    // Event "A_zdown_c_on".
    IF NOT progress THEN
        b1 := (state0.dvar_M_sup_A_zdown) = (elit_Off);
        b1 := b1 AND ((state0.dvar_M_sup_sup) = (elit_X));
        IF b1 THEN
            b3 := (state0.dvar_M_sup_A_x2distributing) = (elit_On);
            b3 := b3 AND ((state0.dvar_M_sup_A_x2testing) = (elit_On));
            b3 := b3 AND ((state0.dvar_M_sup_S_Hinitialized) = (elit_On));
            b3 := b3 AND ((state0.dvar_M_sup_S_product4) = (elit_On));
            b3 := b3 AND ((state0.dvar_M_sup_S_product1) = (elit_On));
            b3 := b3 AND ((state0.dvar_M_sup_S_product2) = (elit_On));
            b3 := b3 AND ((state0.dvar_M_sup_S_product3) = (elit_On));
            b3 := b3 AND ((state0.dvar_M_sup_S_gripper) = (elit_Off));
            b3 := b3 AND ((state0.dvar_M_sup_S_xpos_at3) = (elit_On));
            b3 := b3 AND ((state0.dvar_M_sup_S_zpos_atup) = (elit_On));
            b2 := b3;
            IF NOT(b2) THEN
                b3 := (state0.dvar_M_sup_A_x2distributing) = (elit_On);
                b3 := b3 AND ((state0.dvar_M_sup_A_x2testing) = (elit_On));
                b3 := b3 AND ((state0.dvar_M_sup_S_Hinitialized) = (elit_On));
                b3 := b3 AND ((state0.dvar_M_sup_S_product4) = (elit_On));
                b3 := b3 AND ((state0.dvar_M_sup_S_product1) = (elit_On));
                b3 := b3 AND ((state0.dvar_M_sup_S_product2) = (elit_On));
                b3 := b3 AND ((state0.dvar_M_sup_S_product3) = (elit_On));
                b3 := b3 AND ((state0.dvar_M_sup_S_gripper) = (elit_Off));
                b3 := b3 AND ((state0.dvar_M_sup_S_xpos_at3) = (elit_Off));
                b3 := b3 AND ((state0.dvar_M_sup_S_xpos_at2) = (elit_On));
                b3 := b3 AND ((state0.dvar_M_sup_S_zpos_atup) = (elit_On));
                b2 := b2 OR (b3);
            END_IF;
            IF NOT(b2) THEN
                b3 := (state0.dvar_M_sup_A_x2distributing) = (elit_On);
                b3 := b3 AND ((state0.dvar_M_sup_A_x2testing) = (elit_On));
                b3 := b3 AND ((state0.dvar_M_sup_S_Hinitialized) = (elit_On));
                b3 := b3 AND ((state0.dvar_M_sup_S_product4) = (elit_On));
                b3 := b3 AND ((state0.dvar_M_sup_S_product1) = (elit_On));
                b3 := b3 AND ((state0.dvar_M_sup_S_product2) = (elit_On));
                b3 := b3 AND ((state0.dvar_M_sup_S_product3) = (elit_On));
                b3 := b3 AND ((state0.dvar_M_sup_S_gripper) = (elit_Off));
                b3 := b3 AND ((state0.dvar_M_sup_S_xpos_at3) = (elit_Off));
                b3 := b3 AND ((state0.dvar_M_sup_S_xpos_at2) = (elit_Off));
                b3 := b3 AND ((state0.dvar_M_sup_S_xpos_at1) = (elit_On));
                b3 := b3 AND ((state0.dvar_M_sup_S_zpos_atup) = (elit_On));
                b2 := b2 OR (b3);
            END_IF;
            IF NOT(b2) THEN
                b3 := (state0.dvar_M_sup_A_x2distributing) = (elit_On);
                b3 := b3 AND ((state0.dvar_M_sup_A_x2testing) = (elit_On));
                b3 := b3 AND ((state0.dvar_M_sup_S_Hinitialized) = (elit_On));
                b3 := b3 AND ((state0.dvar_M_sup_S_product4) = (elit_On));
                b3 := b3 AND ((state0.dvar_M_sup_S_product1) = (elit_On));
                b3 := b3 AND ((state0.dvar_M_sup_S_product2) = (elit_On));
                b3 := b3 AND ((state0.dvar_M_sup_S_product3) = (elit_Off));
                b3 := b3 AND ((state0.dvar_M_sup_S_gripper) = (elit_Off));
                b3 := b3 AND ((state0.dvar_M_sup_S_xpos_at2) = (elit_On));
                b3 := b3 AND ((state0.dvar_M_sup_S_zpos_atup) = (elit_On));
                b2 := b2 OR (b3);
            END_IF;
            IF NOT(b2) THEN
                b3 := (state0.dvar_M_sup_A_x2distributing) = (elit_On);
                b3 := b3 AND ((state0.dvar_M_sup_A_x2testing) = (elit_On));
                b3 := b3 AND ((state0.dvar_M_sup_S_Hinitialized) = (elit_On));
                b3 := b3 AND ((state0.dvar_M_sup_S_product4) = (elit_On));
                b3 := b3 AND ((state0.dvar_M_sup_S_product1) = (elit_On));
                b3 := b3 AND ((state0.dvar_M_sup_S_product2) = (elit_On));
                b3 := b3 AND ((state0.dvar_M_sup_S_product3) = (elit_Off));
                b3 := b3 AND ((state0.dvar_M_sup_S_gripper) = (elit_Off));
                b3 := b3 AND ((state0.dvar_M_sup_S_xpos_at2) = (elit_Off));
                b3 := b3 AND ((state0.dvar_M_sup_S_xpos_at1) = (elit_On));
                b3 := b3 AND ((state0.dvar_M_sup_S_zpos_atup) = (elit_On));
                b2 := b2 OR (b3);
            END_IF;
            IF NOT(b2) THEN
                b3 := (state0.dvar_M_sup_A_x2distributing) = (elit_On);
                b3 := b3 AND ((state0.dvar_M_sup_A_x2testing) = (elit_On));
                b3 := b3 AND ((state0.dvar_M_sup_S_Hinitialized) = (elit_On));
                b3 := b3 AND ((state0.dvar_M_sup_S_product4) = (elit_On));
                b3 := b3 AND ((state0.dvar_M_sup_S_product1) = (elit_On));
                b3 := b3 AND ((state0.dvar_M_sup_S_product2) = (elit_Off));
                b3 := b3 AND ((state0.dvar_M_sup_S_product3) = (elit_On));
                b3 := b3 AND ((state0.dvar_M_sup_S_gripper) = (elit_Off));
                b3 := b3 AND ((state0.dvar_M_sup_S_xpos_at3) = (elit_On));
                b3 := b3 AND ((state0.dvar_M_sup_S_zpos_atup) = (elit_On));
                b2 := b2 OR (b3);
            END_IF;
            IF NOT(b2) THEN
                b3 := (state0.dvar_M_sup_A_x2distributing) = (elit_On);
                b3 := b3 AND ((state0.dvar_M_sup_A_x2testing) = (elit_On));
                b3 := b3 AND ((state0.dvar_M_sup_S_Hinitialized) = (elit_On));
                b3 := b3 AND ((state0.dvar_M_sup_S_product4) = (elit_On));
                b3 := b3 AND ((state0.dvar_M_sup_S_product1) = (elit_On));
                b3 := b3 AND ((state0.dvar_M_sup_S_product2) = (elit_Off));
                b3 := b3 AND ((state0.dvar_M_sup_S_product3) = (elit_On));
                b3 := b3 AND ((state0.dvar_M_sup_S_gripper) = (elit_Off));
                b3 := b3 AND ((state0.dvar_M_sup_S_xpos_at3) = (elit_Off));
                b3 := b3 AND ((state0.dvar_M_sup_S_xpos_at1) = (elit_On));
                b3 := b3 AND ((state0.dvar_M_sup_S_zpos_atup) = (elit_On));
                b2 := b2 OR (b3);
            END_IF;
            IF NOT(b2) THEN
                b3 := (state0.dvar_M_sup_A_x2distributing) = (elit_On);
                b3 := b3 AND ((state0.dvar_M_sup_A_x2testing) = (elit_On));
                b3 := b3 AND ((state0.dvar_M_sup_S_Hinitialized) = (elit_On));
                b3 := b3 AND ((state0.dvar_M_sup_S_product4) = (elit_On));
                b3 := b3 AND ((state0.dvar_M_sup_S_product1) = (elit_On));
                b3 := b3 AND ((state0.dvar_M_sup_S_product2) = (elit_Off));
                b3 := b3 AND ((state0.dvar_M_sup_S_product3) = (elit_Off));
                b3 := b3 AND ((state0.dvar_M_sup_S_gripper) = (elit_Off));
                b3 := b3 AND ((state0.dvar_M_sup_S_xpos_at1) = (elit_On));
                b3 := b3 AND ((state0.dvar_M_sup_S_zpos_atup) = (elit_On));
                b2 := b2 OR (b3);
            END_IF;
            IF NOT(b2) THEN
                b3 := (state0.dvar_M_sup_A_x2distributing) = (elit_On);
                b3 := b3 AND ((state0.dvar_M_sup_A_x2testing) = (elit_On));
                b3 := b3 AND ((state0.dvar_M_sup_S_Hinitialized) = (elit_On));
                b3 := b3 AND ((state0.dvar_M_sup_S_product4) = (elit_On));
                b3 := b3 AND ((state0.dvar_M_sup_S_product1) = (elit_Off));
                b3 := b3 AND ((state0.dvar_M_sup_S_product2) = (elit_On));
                b3 := b3 AND ((state0.dvar_M_sup_S_product3) = (elit_On));
                b3 := b3 AND ((state0.dvar_M_sup_S_gripper) = (elit_Off));
                b3 := b3 AND ((state0.dvar_M_sup_S_xpos_at3) = (elit_On));
                b3 := b3 AND ((state0.dvar_M_sup_S_zpos_atup) = (elit_On));
                b2 := b2 OR (b3);
            END_IF;
            IF NOT(b2) THEN
                b3 := (state0.dvar_M_sup_A_x2distributing) = (elit_On);
                b3 := b3 AND ((state0.dvar_M_sup_A_x2testing) = (elit_On));
                b3 := b3 AND ((state0.dvar_M_sup_S_Hinitialized) = (elit_On));
                b3 := b3 AND ((state0.dvar_M_sup_S_product4) = (elit_On));
                b3 := b3 AND ((state0.dvar_M_sup_S_product1) = (elit_Off));
                b3 := b3 AND ((state0.dvar_M_sup_S_product2) = (elit_On));
                b3 := b3 AND ((state0.dvar_M_sup_S_product3) = (elit_On));
                b3 := b3 AND ((state0.dvar_M_sup_S_gripper) = (elit_Off));
                b3 := b3 AND ((state0.dvar_M_sup_S_xpos_at3) = (elit_Off));
                b3 := b3 AND ((state0.dvar_M_sup_S_xpos_at2) = (elit_On));
                b3 := b3 AND ((state0.dvar_M_sup_S_zpos_atup) = (elit_On));
                b2 := b2 OR (b3);
            END_IF;
            IF NOT(b2) THEN
                b3 := (state0.dvar_M_sup_A_x2distributing) = (elit_On);
                b3 := b3 AND ((state0.dvar_M_sup_A_x2testing) = (elit_On));
                b3 := b3 AND ((state0.dvar_M_sup_S_Hinitialized) = (elit_On));
                b3 := b3 AND ((state0.dvar_M_sup_S_product4) = (elit_On));
                b3 := b3 AND ((state0.dvar_M_sup_S_product1) = (elit_Off));
                b3 := b3 AND ((state0.dvar_M_sup_S_product2) = (elit_On));
                b3 := b3 AND ((state0.dvar_M_sup_S_product3) = (elit_Off));
                b3 := b3 AND ((state0.dvar_M_sup_S_gripper) = (elit_Off));
                b3 := b3 AND ((state0.dvar_M_sup_S_xpos_at2) = (elit_On));
                b3 := b3 AND ((state0.dvar_M_sup_S_zpos_atup) = (elit_On));
                b2 := b2 OR (b3);
            END_IF;
            IF NOT(b2) THEN
                b3 := (state0.dvar_M_sup_A_x2distributing) = (elit_On);
                b3 := b3 AND ((state0.dvar_M_sup_A_x2testing) = (elit_On));
                b3 := b3 AND ((state0.dvar_M_sup_S_Hinitialized) = (elit_On));
                b3 := b3 AND ((state0.dvar_M_sup_S_product4) = (elit_On));
                b3 := b3 AND ((state0.dvar_M_sup_S_product1) = (elit_Off));
                b3 := b3 AND ((state0.dvar_M_sup_S_product2) = (elit_Off));
                b3 := b3 AND ((state0.dvar_M_sup_S_product3) = (elit_On));
                b3 := b3 AND ((state0.dvar_M_sup_S_gripper) = (elit_Off));
                b3 := b3 AND ((state0.dvar_M_sup_S_xpos_at3) = (elit_On));
                b3 := b3 AND ((state0.dvar_M_sup_S_zpos_atup) = (elit_On));
                b2 := b2 OR (b3);
            END_IF;
            IF NOT(b2) THEN
                b3 := (state0.dvar_M_sup_A_x2distributing) = (elit_On);
                b3 := b3 AND ((state0.dvar_M_sup_A_x2testing) = (elit_On));
                b3 := b3 AND ((state0.dvar_M_sup_S_Hinitialized) = (elit_On));
                b3 := b3 AND ((state0.dvar_M_sup_S_product4) = (elit_Off));
                b3 := b3 AND ((state0.dvar_M_sup_S_product1) = (elit_On));
                b3 := b3 AND ((state0.dvar_M_sup_S_product2) = (elit_On));
                b3 := b3 AND ((state0.dvar_M_sup_S_product3) = (elit_On));
                b3 := b3 AND ((state0.dvar_M_sup_S_gripper) = (elit_On));
                b3 := b3 AND ((state0.dvar_M_sup_S_xpos_atdrop) = (elit_On));
                b3 := b3 AND ((state0.dvar_M_sup_S_zpos_atup) = (elit_On));
                b2 := b2 OR (b3);
            END_IF;
            IF NOT(b2) THEN
                b3 := (state0.dvar_M_sup_A_x2distributing) = (elit_On);
                b3 := b3 AND ((state0.dvar_M_sup_A_x2testing) = (elit_On));
                b3 := b3 AND ((state0.dvar_M_sup_S_Hinitialized) = (elit_On));
                b3 := b3 AND ((state0.dvar_M_sup_S_product4) = (elit_Off));
                b3 := b3 AND ((state0.dvar_M_sup_S_product1) = (elit_On));
                b3 := b3 AND ((state0.dvar_M_sup_S_product2) = (elit_On));
                b3 := b3 AND ((state0.dvar_M_sup_S_product3) = (elit_On));
                b3 := b3 AND ((state0.dvar_M_sup_S_gripper) = (elit_Off));
                b3 := b3 AND ((state0.dvar_M_sup_S_xpos_at3) = (elit_On));
                b3 := b3 AND ((state0.dvar_M_sup_S_zpos_atup) = (elit_On));
                b2 := b2 OR (b3);
            END_IF;
            IF NOT(b2) THEN
                b3 := (state0.dvar_M_sup_A_x2distributing) = (elit_On);
                b3 := b3 AND ((state0.dvar_M_sup_A_x2testing) = (elit_On));
                b3 := b3 AND ((state0.dvar_M_sup_S_Hinitialized) = (elit_On));
                b3 := b3 AND ((state0.dvar_M_sup_S_product4) = (elit_Off));
                b3 := b3 AND ((state0.dvar_M_sup_S_product1) = (elit_On));
                b3 := b3 AND ((state0.dvar_M_sup_S_product2) = (elit_On));
                b3 := b3 AND ((state0.dvar_M_sup_S_product3) = (elit_On));
                b3 := b3 AND ((state0.dvar_M_sup_S_gripper) = (elit_Off));
                b3 := b3 AND ((state0.dvar_M_sup_S_xpos_at3) = (elit_Off));
                b3 := b3 AND ((state0.dvar_M_sup_S_xpos_at2) = (elit_On));
                b3 := b3 AND ((state0.dvar_M_sup_S_zpos_atup) = (elit_On));
                b2 := b2 OR (b3);
            END_IF;
            IF NOT(b2) THEN
                b3 := (state0.dvar_M_sup_A_x2distributing) = (elit_On);
                b3 := b3 AND ((state0.dvar_M_sup_A_x2testing) = (elit_On));
                b3 := b3 AND ((state0.dvar_M_sup_S_Hinitialized) = (elit_On));
                b3 := b3 AND ((state0.dvar_M_sup_S_product4) = (elit_Off));
                b3 := b3 AND ((state0.dvar_M_sup_S_product1) = (elit_On));
                b3 := b3 AND ((state0.dvar_M_sup_S_product2) = (elit_On));
                b3 := b3 AND ((state0.dvar_M_sup_S_product3) = (elit_On));
                b3 := b3 AND ((state0.dvar_M_sup_S_gripper) = (elit_Off));
                b3 := b3 AND ((state0.dvar_M_sup_S_xpos_at3) = (elit_Off));
                b3 := b3 AND ((state0.dvar_M_sup_S_xpos_at2) = (elit_Off));
                b3 := b3 AND ((state0.dvar_M_sup_S_xpos_at1) = (elit_On));
                b3 := b3 AND ((state0.dvar_M_sup_S_zpos_atup) = (elit_On));
                b2 := b2 OR (b3);
            END_IF;
            IF NOT(b2) THEN
                b3 := (state0.dvar_M_sup_A_x2distributing) = (elit_On);
                b3 := b3 AND ((state0.dvar_M_sup_A_x2testing) = (elit_On));
                b3 := b3 AND ((state0.dvar_M_sup_S_Hinitialized) = (elit_On));
                b3 := b3 AND ((state0.dvar_M_sup_S_product4) = (elit_Off));
                b3 := b3 AND ((state0.dvar_M_sup_S_product1) = (elit_On));
                b3 := b3 AND ((state0.dvar_M_sup_S_product2) = (elit_On));
                b3 := b3 AND ((state0.dvar_M_sup_S_product3) = (elit_Off));
                b3 := b3 AND ((state0.dvar_M_sup_S_gripper) = (elit_On));
                b3 := b3 AND ((state0.dvar_M_sup_S_xpos_atdrop) = (elit_On));
                b3 := b3 AND ((state0.dvar_M_sup_S_zpos_atup) = (elit_On));
                b2 := b2 OR (b3);
            END_IF;
            IF NOT(b2) THEN
                b3 := (state0.dvar_M_sup_A_x2distributing) = (elit_On);
                b3 := b3 AND ((state0.dvar_M_sup_A_x2testing) = (elit_On));
                b3 := b3 AND ((state0.dvar_M_sup_S_Hinitialized) = (elit_On));
                b3 := b3 AND ((state0.dvar_M_sup_S_product4) = (elit_Off));
                b3 := b3 AND ((state0.dvar_M_sup_S_product1) = (elit_On));
                b3 := b3 AND ((state0.dvar_M_sup_S_product2) = (elit_On));
                b3 := b3 AND ((state0.dvar_M_sup_S_product3) = (elit_Off));
                b3 := b3 AND ((state0.dvar_M_sup_S_gripper) = (elit_Off));
                b3 := b3 AND ((state0.dvar_M_sup_S_xpos_at2) = (elit_On));
                b3 := b3 AND ((state0.dvar_M_sup_S_zpos_atup) = (elit_On));
                b2 := b2 OR (b3);
            END_IF;
            IF NOT(b2) THEN
                b3 := (state0.dvar_M_sup_A_x2distributing) = (elit_On);
                b3 := b3 AND ((state0.dvar_M_sup_A_x2testing) = (elit_On));
                b3 := b3 AND ((state0.dvar_M_sup_S_Hinitialized) = (elit_On));
                b3 := b3 AND ((state0.dvar_M_sup_S_product4) = (elit_Off));
                b3 := b3 AND ((state0.dvar_M_sup_S_product1) = (elit_On));
                b3 := b3 AND ((state0.dvar_M_sup_S_product2) = (elit_On));
                b3 := b3 AND ((state0.dvar_M_sup_S_product3) = (elit_Off));
                b3 := b3 AND ((state0.dvar_M_sup_S_gripper) = (elit_Off));
                b3 := b3 AND ((state0.dvar_M_sup_S_xpos_at2) = (elit_Off));
                b3 := b3 AND ((state0.dvar_M_sup_S_xpos_at1) = (elit_On));
                b3 := b3 AND ((state0.dvar_M_sup_S_zpos_atup) = (elit_On));
                b2 := b2 OR (b3);
            END_IF;
            IF NOT(b2) THEN
                b3 := (state0.dvar_M_sup_A_x2distributing) = (elit_On);
                b3 := b3 AND ((state0.dvar_M_sup_A_x2testing) = (elit_On));
                b3 := b3 AND ((state0.dvar_M_sup_S_Hinitialized) = (elit_On));
                b3 := b3 AND ((state0.dvar_M_sup_S_product4) = (elit_Off));
                b3 := b3 AND ((state0.dvar_M_sup_S_product1) = (elit_On));
                b3 := b3 AND ((state0.dvar_M_sup_S_product2) = (elit_Off));
                b3 := b3 AND ((state0.dvar_M_sup_S_product3) = (elit_On));
                b3 := b3 AND ((state0.dvar_M_sup_S_gripper) = (elit_On));
                b3 := b3 AND ((state0.dvar_M_sup_S_xpos_atdrop) = (elit_On));
                b3 := b3 AND ((state0.dvar_M_sup_S_zpos_atup) = (elit_On));
                b2 := b2 OR (b3);
            END_IF;
            IF NOT(b2) THEN
                b3 := (state0.dvar_M_sup_A_x2distributing) = (elit_On);
                b3 := b3 AND ((state0.dvar_M_sup_A_x2testing) = (elit_On));
                b3 := b3 AND ((state0.dvar_M_sup_S_Hinitialized) = (elit_On));
                b3 := b3 AND ((state0.dvar_M_sup_S_product4) = (elit_Off));
                b3 := b3 AND ((state0.dvar_M_sup_S_product1) = (elit_On));
                b3 := b3 AND ((state0.dvar_M_sup_S_product2) = (elit_Off));
                b3 := b3 AND ((state0.dvar_M_sup_S_product3) = (elit_On));
                b3 := b3 AND ((state0.dvar_M_sup_S_gripper) = (elit_Off));
                b3 := b3 AND ((state0.dvar_M_sup_S_xpos_at3) = (elit_On));
                b3 := b3 AND ((state0.dvar_M_sup_S_zpos_atup) = (elit_On));
                b2 := b2 OR (b3);
            END_IF;
            IF NOT(b2) THEN
                b3 := (state0.dvar_M_sup_A_x2distributing) = (elit_On);
                b3 := b3 AND ((state0.dvar_M_sup_A_x2testing) = (elit_On));
                b3 := b3 AND ((state0.dvar_M_sup_S_Hinitialized) = (elit_On));
                b3 := b3 AND ((state0.dvar_M_sup_S_product4) = (elit_Off));
                b3 := b3 AND ((state0.dvar_M_sup_S_product1) = (elit_On));
                b3 := b3 AND ((state0.dvar_M_sup_S_product2) = (elit_Off));
                b3 := b3 AND ((state0.dvar_M_sup_S_product3) = (elit_On));
                b3 := b3 AND ((state0.dvar_M_sup_S_gripper) = (elit_Off));
                b3 := b3 AND ((state0.dvar_M_sup_S_xpos_at3) = (elit_Off));
                b3 := b3 AND ((state0.dvar_M_sup_S_xpos_at1) = (elit_On));
                b3 := b3 AND ((state0.dvar_M_sup_S_zpos_atup) = (elit_On));
                b2 := b2 OR (b3);
            END_IF;
            IF NOT(b2) THEN
                b3 := (state0.dvar_M_sup_A_x2distributing) = (elit_On);
                b3 := b3 AND ((state0.dvar_M_sup_A_x2testing) = (elit_On));
                b3 := b3 AND ((state0.dvar_M_sup_S_Hinitialized) = (elit_On));
                b3 := b3 AND ((state0.dvar_M_sup_S_product4) = (elit_Off));
                b3 := b3 AND ((state0.dvar_M_sup_S_product1) = (elit_On));
                b3 := b3 AND ((state0.dvar_M_sup_S_product2) = (elit_Off));
                b3 := b3 AND ((state0.dvar_M_sup_S_product3) = (elit_Off));
                b3 := b3 AND ((state0.dvar_M_sup_S_gripper) = (elit_On));
                b3 := b3 AND ((state0.dvar_M_sup_S_xpos_atdrop) = (elit_On));
                b3 := b3 AND ((state0.dvar_M_sup_S_zpos_atup) = (elit_On));
                b2 := b2 OR (b3);
            END_IF;
            IF NOT(b2) THEN
                b3 := (state0.dvar_M_sup_A_x2distributing) = (elit_On);
                b3 := b3 AND ((state0.dvar_M_sup_A_x2testing) = (elit_On));
                b3 := b3 AND ((state0.dvar_M_sup_S_Hinitialized) = (elit_On));
                b3 := b3 AND ((state0.dvar_M_sup_S_product4) = (elit_Off));
                b3 := b3 AND ((state0.dvar_M_sup_S_product1) = (elit_On));
                b3 := b3 AND ((state0.dvar_M_sup_S_product2) = (elit_Off));
                b3 := b3 AND ((state0.dvar_M_sup_S_product3) = (elit_Off));
                b3 := b3 AND ((state0.dvar_M_sup_S_gripper) = (elit_Off));
                b3 := b3 AND ((state0.dvar_M_sup_S_xpos_at1) = (elit_On));
                b3 := b3 AND ((state0.dvar_M_sup_S_zpos_atup) = (elit_On));
                b2 := b2 OR (b3);
            END_IF;
            IF NOT(b2) THEN
                b3 := (state0.dvar_M_sup_A_x2distributing) = (elit_On);
                b3 := b3 AND ((state0.dvar_M_sup_A_x2testing) = (elit_On));
                b3 := b3 AND ((state0.dvar_M_sup_S_Hinitialized) = (elit_On));
                b3 := b3 AND ((state0.dvar_M_sup_S_product4) = (elit_Off));
                b3 := b3 AND ((state0.dvar_M_sup_S_product1) = (elit_Off));
                b3 := b3 AND ((state0.dvar_M_sup_S_product2) = (elit_On));
                b3 := b3 AND ((state0.dvar_M_sup_S_product3) = (elit_On));
                b3 := b3 AND ((state0.dvar_M_sup_S_gripper) = (elit_On));
                b3 := b3 AND ((state0.dvar_M_sup_S_xpos_atdrop) = (elit_On));
                b3 := b3 AND ((state0.dvar_M_sup_S_zpos_atup) = (elit_On));
                b2 := b2 OR (b3);
            END_IF;
            IF NOT(b2) THEN
                b3 := (state0.dvar_M_sup_A_x2distributing) = (elit_On);
                b3 := b3 AND ((state0.dvar_M_sup_A_x2testing) = (elit_On));
                b3 := b3 AND ((state0.dvar_M_sup_S_Hinitialized) = (elit_On));
                b3 := b3 AND ((state0.dvar_M_sup_S_product4) = (elit_Off));
                b3 := b3 AND ((state0.dvar_M_sup_S_product1) = (elit_Off));
                b3 := b3 AND ((state0.dvar_M_sup_S_product2) = (elit_On));
                b3 := b3 AND ((state0.dvar_M_sup_S_product3) = (elit_On));
                b3 := b3 AND ((state0.dvar_M_sup_S_gripper) = (elit_Off));
                b3 := b3 AND ((state0.dvar_M_sup_S_xpos_at3) = (elit_On));
                b3 := b3 AND ((state0.dvar_M_sup_S_zpos_atup) = (elit_On));
                b2 := b2 OR (b3);
            END_IF;
            IF NOT(b2) THEN
                b3 := (state0.dvar_M_sup_A_x2distributing) = (elit_On);
                b3 := b3 AND ((state0.dvar_M_sup_A_x2testing) = (elit_On));
                b3 := b3 AND ((state0.dvar_M_sup_S_Hinitialized) = (elit_On));
                b3 := b3 AND ((state0.dvar_M_sup_S_product4) = (elit_Off));
                b3 := b3 AND ((state0.dvar_M_sup_S_product1) = (elit_Off));
                b3 := b3 AND ((state0.dvar_M_sup_S_product2) = (elit_On));
                b3 := b3 AND ((state0.dvar_M_sup_S_product3) = (elit_On));
                b3 := b3 AND ((state0.dvar_M_sup_S_gripper) = (elit_Off));
                b3 := b3 AND ((state0.dvar_M_sup_S_xpos_at3) = (elit_Off));
                b3 := b3 AND ((state0.dvar_M_sup_S_xpos_at2) = (elit_On));
                b3 := b3 AND ((state0.dvar_M_sup_S_zpos_atup) = (elit_On));
                b2 := b2 OR (b3);
            END_IF;
            IF NOT(b2) THEN
                b3 := (state0.dvar_M_sup_A_x2distributing) = (elit_On);
                b3 := b3 AND ((state0.dvar_M_sup_A_x2testing) = (elit_On));
                b3 := b3 AND ((state0.dvar_M_sup_S_Hinitialized) = (elit_On));
                b3 := b3 AND ((state0.dvar_M_sup_S_product4) = (elit_Off));
                b3 := b3 AND ((state0.dvar_M_sup_S_product1) = (elit_Off));
                b3 := b3 AND ((state0.dvar_M_sup_S_product2) = (elit_On));
                b3 := b3 AND ((state0.dvar_M_sup_S_product3) = (elit_Off));
                b3 := b3 AND ((state0.dvar_M_sup_S_gripper) = (elit_On));
                b3 := b3 AND ((state0.dvar_M_sup_S_xpos_atdrop) = (elit_On));
                b3 := b3 AND ((state0.dvar_M_sup_S_zpos_atup) = (elit_On));
                b2 := b2 OR (b3);
            END_IF;
            IF NOT(b2) THEN
                b3 := (state0.dvar_M_sup_A_x2distributing) = (elit_On);
                b3 := b3 AND ((state0.dvar_M_sup_A_x2testing) = (elit_On));
                b3 := b3 AND ((state0.dvar_M_sup_S_Hinitialized) = (elit_On));
                b3 := b3 AND ((state0.dvar_M_sup_S_product4) = (elit_Off));
                b3 := b3 AND ((state0.dvar_M_sup_S_product1) = (elit_Off));
                b3 := b3 AND ((state0.dvar_M_sup_S_product2) = (elit_On));
                b3 := b3 AND ((state0.dvar_M_sup_S_product3) = (elit_Off));
                b3 := b3 AND ((state0.dvar_M_sup_S_gripper) = (elit_Off));
                b3 := b3 AND ((state0.dvar_M_sup_S_xpos_at2) = (elit_On));
                b3 := b3 AND ((state0.dvar_M_sup_S_zpos_atup) = (elit_On));
                b2 := b2 OR (b3);
            END_IF;
            IF NOT(b2) THEN
                b3 := (state0.dvar_M_sup_A_x2distributing) = (elit_On);
                b3 := b3 AND ((state0.dvar_M_sup_A_x2testing) = (elit_On));
                b3 := b3 AND ((state0.dvar_M_sup_S_Hinitialized) = (elit_On));
                b3 := b3 AND ((state0.dvar_M_sup_S_product4) = (elit_Off));
                b3 := b3 AND ((state0.dvar_M_sup_S_product1) = (elit_Off));
                b3 := b3 AND ((state0.dvar_M_sup_S_product2) = (elit_Off));
                b3 := b3 AND ((state0.dvar_M_sup_S_product3) = (elit_On));
                b3 := b3 AND ((state0.dvar_M_sup_S_gripper) = (elit_On));
                b3 := b3 AND ((state0.dvar_M_sup_S_xpos_atdrop) = (elit_On));
                b3 := b3 AND ((state0.dvar_M_sup_S_zpos_atup) = (elit_On));
                b2 := b2 OR (b3);
            END_IF;
            IF NOT(b2) THEN
                b3 := (state0.dvar_M_sup_A_x2distributing) = (elit_On);
                b3 := b3 AND ((state0.dvar_M_sup_A_x2testing) = (elit_On));
                b3 := b3 AND ((state0.dvar_M_sup_S_Hinitialized) = (elit_On));
                b3 := b3 AND ((state0.dvar_M_sup_S_product4) = (elit_Off));
                b3 := b3 AND ((state0.dvar_M_sup_S_product1) = (elit_Off));
                b3 := b3 AND ((state0.dvar_M_sup_S_product2) = (elit_Off));
                b3 := b3 AND ((state0.dvar_M_sup_S_product3) = (elit_On));
                b3 := b3 AND ((state0.dvar_M_sup_S_gripper) = (elit_Off));
                b3 := b3 AND ((state0.dvar_M_sup_S_xpos_at3) = (elit_On));
                b3 := b3 AND ((state0.dvar_M_sup_S_zpos_atup) = (elit_On));
                b2 := b2 OR (b3);
            END_IF;
            IF NOT(b2) THEN
                b3 := (state0.dvar_M_sup_A_x2distributing) = (elit_On);
                b3 := b3 AND ((state0.dvar_M_sup_A_x2testing) = (elit_On));
                b3 := b3 AND ((state0.dvar_M_sup_S_Hinitialized) = (elit_On));
                b3 := b3 AND ((state0.dvar_M_sup_S_product4) = (elit_Off));
                b3 := b3 AND ((state0.dvar_M_sup_S_product1) = (elit_Off));
                b3 := b3 AND ((state0.dvar_M_sup_S_product2) = (elit_Off));
                b3 := b3 AND ((state0.dvar_M_sup_S_product3) = (elit_Off));
                b3 := b3 AND ((state0.dvar_M_sup_S_gripper) = (elit_On));
                b3 := b3 AND ((state0.dvar_M_sup_S_xpos_atdrop) = (elit_On));
                b3 := b3 AND ((state0.dvar_M_sup_S_zpos_atup) = (elit_On));
                b2 := b2 OR (b3);
            END_IF;
            b1 := b1 AND (b2);
        END_IF;
        IF b1 THEN
            progress := TRUE;
            state1 := state0;

            state1.dvar_M_sup_A_zdown := elit_On;

            state0 := state1;
        END_IF;
    END_IF;

    // Event "BTimer_c_on".
    IF NOT progress THEN
        b1 := (state0.dvar_M_BTimer1) = (elit_Off);
        b1 := b1 AND ((state0.dvar_M_sup_BTimer) = (elit_Off));
        b1 := b1 AND ((state0.dvar_M_sup_sup) = (elit_X));
        b1 := b1 AND ((state0.dvar_M_sup_S_atend) = (elit_On));
        IF b1 THEN
            progress := TRUE;
            state1 := state0;

            state1.dvar_M_BTimer1 := elit_Running;
            state1.dvar_M_sup_BTimer := elit_Running;

            state0 := state1;
        END_IF;
    END_IF;

    // Event "BTimer_c_reset".
    IF NOT progress THEN
        b2 := (state0.dvar_M_BTimer1) = (elit_Running);
        b2 := b2 OR ((state0.dvar_M_BTimer1) = (elit_Timeout));
        b1 := b2;
        IF b1 THEN
            b2 := (state0.dvar_M_sup_BTimer) = (elit_Running);
            b2 := b2 OR ((state0.dvar_M_sup_BTimer) = (elit_Timeout));
            b1 := b1 AND (b2);
        END_IF;
        b1 := b1 AND ((state0.dvar_M_sup_sup) = (elit_X));
        IF b1 THEN
            b2 := (state0.dvar_M_sup_A_conveyerB) = (elit_Off);
            b2 := b2 OR ((state0.dvar_M_sup_S_atin) = (elit_On));
            b1 := b1 AND (b2);
        END_IF;
        IF b1 THEN
            progress := TRUE;
            state1 := state0;

            IF ((state0.dvar_M_BTimer1) = (elit_Running)) THEN
                state1.cvar_M_BTimer1_t := 0.0;
                state1.dvar_M_BTimer1 := elit_Off;
            ELSIF ((state0.dvar_M_BTimer1) = (elit_Timeout)) THEN
                state1.cvar_M_BTimer1_t := 0.0;
                state1.dvar_M_BTimer1 := elit_Off;
            END_IF;
            IF ((state0.dvar_M_sup_BTimer) = (elit_Running)) THEN
                state1.dvar_M_sup_BTimer := elit_Off;
            ELSIF ((state0.dvar_M_sup_BTimer) = (elit_Timeout)) THEN
                state1.dvar_M_sup_BTimer := elit_Off;
            END_IF;

            state0 := state1;
        END_IF;
    END_IF;

    // Event "BTimer_u_timeout".
    IF NOT progress THEN
        b1 := (state0.dvar_M_BTimer1) = (elit_Running);
        b1 := b1 AND ((state0.cvar_M_BTimer1_t) > (0.5));
        b1 := b1 AND ((state0.dvar_M_sup_BTimer) = (elit_Running));
        IF b1 THEN
            progress := TRUE;
            state1 := state0;

            state1.dvar_M_BTimer1 := elit_Timeout;
            state1.dvar_M_sup_BTimer := elit_Timeout;

            state0 := state1;
        END_IF;
    END_IF;

    // Event "S_atdrill_u_off".
    IF NOT progress THEN
        b1 := (state0.dvar_M_BoolToEventsP) = (elit_X);
        b1 := b1 AND (NOT(ivar_s_atdrill));
        b1 := b1 AND ((state0.dvar_M_sup_S_atdrill) = (elit_On));
        IF b1 THEN
            progress := TRUE;
            state1 := state0;

            state1.dvar_M_sup_S_atdrill := elit_Off;

            state0 := state1;
        END_IF;
    END_IF;

    // Event "S_atdrill_u_on".
    IF NOT progress THEN
        b1 := (state0.dvar_M_BoolToEventsP) = (elit_X);
        b1 := b1 AND (ivar_s_atdrill);
        b1 := b1 AND ((state0.dvar_M_sup_S_atdrill) = (elit_Off));
        IF b1 THEN
            progress := TRUE;
            state1 := state0;

            state1.dvar_M_sup_S_atdrill := elit_On;

            state0 := state1;
        END_IF;
    END_IF;

    // Event "S_atend_u_off".
    IF NOT progress THEN
        b1 := (state0.dvar_M_BoolToEventsTB) = (elit_X);
        b1 := b1 AND (NOT(ivar_s_atend));
        b1 := b1 AND ((state0.dvar_M_sup_S_atend) = (elit_On));
        IF b1 THEN
            progress := TRUE;
            state1 := state0;

            state1.dvar_M_sup_S_atend := elit_Off;

            state0 := state1;
        END_IF;
    END_IF;

    // Event "S_atend_u_on".
    IF NOT progress THEN
        b1 := (state0.dvar_M_BoolToEventsTB) = (elit_X);
        b1 := b1 AND (ivar_s_atend);
        b1 := b1 AND ((state0.dvar_M_sup_S_atend) = (elit_Off));
        IF b1 THEN
            progress := TRUE;
            state1 := state0;

            state1.dvar_M_sup_S_atend := elit_On;

            state0 := state1;
        END_IF;
    END_IF;

    // Event "S_atexit_u_off".
    IF NOT progress THEN
        b1 := (state0.dvar_M_BoolToEventsP) = (elit_X);
        b1 := b1 AND (NOT(ivar_s_atexit));
        b1 := b1 AND ((state0.dvar_M_sup_S_atexit) = (elit_On));
        IF b1 THEN
            progress := TRUE;
            state1 := state0;

            state1.dvar_M_sup_S_atexit := elit_Off;

            state0 := state1;
        END_IF;
    END_IF;

    // Event "S_atexit_u_on".
    IF NOT progress THEN
        b1 := (state0.dvar_M_BoolToEventsP) = (elit_X);
        b1 := b1 AND (ivar_s_atexit);
        b1 := b1 AND ((state0.dvar_M_sup_S_atexit) = (elit_Off));
        IF b1 THEN
            progress := TRUE;
            state1 := state0;

            state1.dvar_M_sup_S_atexit := elit_On;

            state0 := state1;
        END_IF;
    END_IF;

    // Event "S_atin_u_off".
    IF NOT progress THEN
        b1 := (state0.dvar_M_BoolToEventsTB) = (elit_X);
        b1 := b1 AND (NOT(ivar_s_atin));
        b1 := b1 AND ((state0.dvar_M_sup_S_atin) = (elit_On));
        IF b1 THEN
            progress := TRUE;
            state1 := state0;

            state1.dvar_M_sup_S_atin := elit_Off;

            state0 := state1;
        END_IF;
    END_IF;

    // Event "S_atin_u_on".
    IF NOT progress THEN
        b1 := (state0.dvar_M_BoolToEventsTB) = (elit_X);
        b1 := b1 AND (ivar_s_atin);
        b1 := b1 AND ((state0.dvar_M_sup_S_atin) = (elit_Off));
        IF b1 THEN
            progress := TRUE;
            state1 := state0;

            state1.dvar_M_sup_S_atin := elit_On;

            state0 := state1;
        END_IF;
    END_IF;

    // Event "S_atinput_u_off".
    IF NOT progress THEN
        b1 := (state0.dvar_M_BoolToEventsP) = (elit_X);
        b1 := b1 AND (NOT(ivar_s_atinput));
        b1 := b1 AND ((state0.dvar_M_sup_S_atinput) = (elit_On));
        IF b1 THEN
            progress := TRUE;
            state1 := state0;

            state1.dvar_M_sup_S_atinput := elit_Off;

            state0 := state1;
        END_IF;
    END_IF;

    // Event "S_atinput_u_on".
    IF NOT progress THEN
        b1 := (state0.dvar_M_BoolToEventsP) = (elit_X);
        b1 := b1 AND (ivar_s_atinput);
        b1 := b1 AND ((state0.dvar_M_sup_S_atinput) = (elit_Off));
        IF b1 THEN
            progress := TRUE;
            state1 := state0;

            state1.dvar_M_sup_S_atinput := elit_On;

            state0 := state1;
        END_IF;
    END_IF;

    // Event "S_atseparator_u_off".
    IF NOT progress THEN
        b1 := (state0.dvar_M_BoolToEventsTB) = (elit_X);
        b1 := b1 AND (NOT(ivar_s_atseparator));
        b1 := b1 AND ((state0.dvar_M_sup_S_atseparator) = (elit_On));
        IF b1 THEN
            progress := TRUE;
            state1 := state0;

            state1.dvar_M_sup_S_atseparator := elit_Off;

            state0 := state1;
        END_IF;
    END_IF;

    // Event "S_atseparator_u_on".
    IF NOT progress THEN
        b1 := (state0.dvar_M_BoolToEventsTB) = (elit_X);
        b1 := b1 AND (ivar_s_atseparator);
        b1 := b1 AND ((state0.dvar_M_sup_S_atseparator) = (elit_Off));
        IF b1 THEN
            progress := TRUE;
            state1 := state0;

            state1.dvar_M_sup_S_atseparator := elit_On;

            state0 := state1;
        END_IF;
    END_IF;

    // Event "S_atspare_u_off".
    IF NOT progress THEN
        b1 := (state0.dvar_M_BoolToEventsP) = (elit_X);
        b1 := b1 AND (NOT(ivar_s_atspare));
        b1 := b1 AND ((state0.dvar_M_sup_S_atspare) = (elit_On));
        IF b1 THEN
            progress := TRUE;
            state1 := state0;

            state1.dvar_M_sup_S_atspare := elit_Off;

            state0 := state1;
        END_IF;
    END_IF;

    // Event "S_atspare_u_on".
    IF NOT progress THEN
        b1 := (state0.dvar_M_BoolToEventsP) = (elit_X);
        b1 := b1 AND (ivar_s_atspare);
        b1 := b1 AND ((state0.dvar_M_sup_S_atspare) = (elit_Off));
        IF b1 THEN
            progress := TRUE;
            state1 := state0;

            state1.dvar_M_sup_S_atspare := elit_On;

            state0 := state1;
        END_IF;
    END_IF;

    // Event "S_attest_u_off".
    IF NOT progress THEN
        b1 := (state0.dvar_M_BoolToEventsP) = (elit_X);
        b1 := b1 AND (NOT(ivar_s_attest));
        b1 := b1 AND ((state0.dvar_M_sup_S_attest) = (elit_On));
        IF b1 THEN
            progress := TRUE;
            state1 := state0;

            state1.dvar_M_sup_S_attest := elit_Off;

            state0 := state1;
        END_IF;
    END_IF;

    // Event "S_attest_u_on".
    IF NOT progress THEN
        b1 := (state0.dvar_M_BoolToEventsP) = (elit_X);
        b1 := b1 AND (ivar_s_attest);
        b1 := b1 AND ((state0.dvar_M_sup_S_attest) = (elit_Off));
        IF b1 THEN
            progress := TRUE;
            state1 := state0;

            state1.dvar_M_sup_S_attest := elit_On;

            state0 := state1;
        END_IF;
    END_IF;

    // Event "S_Binitialized_u_off".
    IF NOT progress THEN
        b1 := (state0.dvar_M_BoolToEventsTB) = (elit_X);
        b1 := b1 AND ((state0.dvar_M_HardwareMapTB) <> (elit_initialized));
        b1 := b1 AND ((state0.dvar_M_sup_S_Binitialized) = (elit_On));
        IF b1 THEN
            progress := TRUE;
            state1 := state0;

            state1.dvar_M_sup_S_Binitialized := elit_Off;

            state0 := state1;
        END_IF;
    END_IF;

    // Event "S_Binitialized_u_on".
    IF NOT progress THEN
        b1 := (state0.dvar_M_BoolToEventsTB) = (elit_X);
        b1 := b1 AND ((state0.dvar_M_HardwareMapTB) = (elit_initialized));
        b1 := b1 AND ((state0.dvar_M_sup_S_Binitialized) = (elit_Off));
        IF b1 THEN
            progress := TRUE;
            state1 := state0;

            state1.dvar_M_sup_S_Binitialized := elit_On;

            state0 := state1;
        END_IF;
    END_IF;

    // Event "S_bufferingbusy_u_off".
    IF NOT progress THEN
        b1 := (state0.dvar_M_BoolToEventsTB) = (elit_X);
        b1 := b1 AND (NOT(ivar_s_bufferingbusy));
        b1 := b1 AND ((state0.dvar_M_sup_S_bufferingbusy) = (elit_On));
        IF b1 THEN
            progress := TRUE;
            state1 := state0;

            state1.dvar_M_sup_S_bufferingbusy := elit_Off;

            state0 := state1;
        END_IF;
    END_IF;

    // Event "S_bufferingbusy_u_on".
    IF NOT progress THEN
        b1 := (state0.dvar_M_BoolToEventsTB) = (elit_X);
        b1 := b1 AND (ivar_s_bufferingbusy);
        b1 := b1 AND ((state0.dvar_M_sup_S_bufferingbusy) = (elit_Off));
        IF b1 THEN
            progress := TRUE;
            state1 := state0;

            state1.dvar_M_sup_S_bufferingbusy := elit_On;

            state0 := state1;
        END_IF;
    END_IF;

    // Event "S_capacitive_u_off".
    IF NOT progress THEN
        b1 := (state0.dvar_M_BoolToEventsTB) = (elit_X);
        b1 := b1 AND (NOT(ivar_s_capacitive));
        b1 := b1 AND ((state0.dvar_M_sup_S_capacitive) = (elit_On));
        IF b1 THEN
            progress := TRUE;
            state1 := state0;

            state1.dvar_M_sup_S_capacitive := elit_Off;

            state0 := state1;
        END_IF;
    END_IF;

    // Event "S_capacitive_u_on".
    IF NOT progress THEN
        b1 := (state0.dvar_M_BoolToEventsTB) = (elit_X);
        b1 := b1 AND (ivar_s_capacitive);
        b1 := b1 AND ((state0.dvar_M_sup_S_capacitive) = (elit_Off));
        IF b1 THEN
            progress := TRUE;
            state1 := state0;

            state1.dvar_M_sup_S_capacitive := elit_On;

            state0 := state1;
        END_IF;
    END_IF;

    // Event "S_clamp_u_off".
    IF NOT progress THEN
        b1 := (state0.dvar_M_BoolToEventsP) = (elit_X);
        b1 := b1 AND (NOT(ivar_s_clamp));
        b1 := b1 AND ((state0.dvar_M_sup_S_clamp) = (elit_On));
        IF b1 THEN
            progress := TRUE;
            state1 := state0;

            state1.dvar_M_sup_S_clamp := elit_Off;

            state0 := state1;
        END_IF;
    END_IF;

    // Event "S_clamp_u_on".
    IF NOT progress THEN
        b1 := (state0.dvar_M_BoolToEventsP) = (elit_X);
        b1 := b1 AND (ivar_s_clamp);
        b1 := b1 AND ((state0.dvar_M_sup_S_clamp) = (elit_Off));
        IF b1 THEN
            progress := TRUE;
            state1 := state0;

            state1.dvar_M_sup_S_clamp := elit_On;

            state0 := state1;
        END_IF;
    END_IF;

    // Event "S_Dinitialized_u_off".
    IF NOT progress THEN
        b1 := (state0.dvar_M_BoolToEventsDH) = (elit_X);
        b1 := b1 AND ((state0.dvar_M_HardwareMapDH) <> (elit_initialized));
        b1 := b1 AND ((state0.dvar_M_sup_S_Dinitialized) = (elit_On));
        IF b1 THEN
            progress := TRUE;
            state1 := state0;

            state1.dvar_M_sup_S_Dinitialized := elit_Off;

            state0 := state1;
        END_IF;
    END_IF;

    // Event "S_Dinitialized_u_on".
    IF NOT progress THEN
        b1 := (state0.dvar_M_BoolToEventsDH) = (elit_X);
        b1 := b1 AND ((state0.dvar_M_HardwareMapDH) = (elit_initialized));
        b1 := b1 AND ((state0.dvar_M_sup_S_Dinitialized) = (elit_Off));
        IF b1 THEN
            progress := TRUE;
            state1 := state0;

            state1.dvar_M_sup_S_Dinitialized := elit_On;

            state0 := state1;
        END_IF;
    END_IF;

    // Event "S_drill_down_u_off".
    IF NOT progress THEN
        b1 := (state0.dvar_M_BoolToEventsP) = (elit_X);
        b1 := b1 AND (NOT(ivar_s_drill_down));
        b1 := b1 AND ((state0.dvar_M_sup_S_drill_down) = (elit_On));
        IF b1 THEN
            progress := TRUE;
            state1 := state0;

            state1.dvar_M_sup_S_drill_down := elit_Off;

            state0 := state1;
        END_IF;
    END_IF;

    // Event "S_drill_down_u_on".
    IF NOT progress THEN
        b1 := (state0.dvar_M_BoolToEventsP) = (elit_X);
        b1 := b1 AND (ivar_s_drill_down);
        b1 := b1 AND ((state0.dvar_M_sup_PDynamics) = (elit_X));
        b1 := b1 AND ((state0.dvar_M_sup_S_drill_up) = (elit_Off));
        b1 := b1 AND ((state0.dvar_M_sup_S_drill_down) = (elit_Off));
        IF b1 THEN
            progress := TRUE;
            state1 := state0;

            state1.dvar_M_sup_S_drill_down := elit_On;

            state0 := state1;
        END_IF;
    END_IF;

    // Event "S_drill_up_u_off".
    IF NOT progress THEN
        b1 := (state0.dvar_M_BoolToEventsP) = (elit_X);
        b1 := b1 AND (NOT(ivar_s_drill_up));
        b1 := b1 AND ((state0.dvar_M_sup_S_drill_up) = (elit_On));
        IF b1 THEN
            progress := TRUE;
            state1 := state0;

            state1.dvar_M_sup_S_drill_up := elit_Off;

            state0 := state1;
        END_IF;
    END_IF;

    // Event "S_drill_up_u_on".
    IF NOT progress THEN
        b1 := (state0.dvar_M_BoolToEventsP) = (elit_X);
        b1 := b1 AND (ivar_s_drill_up);
        b1 := b1 AND ((state0.dvar_M_sup_PDynamics) = (elit_X));
        b1 := b1 AND ((state0.dvar_M_sup_S_drill_down) = (elit_Off));
        b1 := b1 AND ((state0.dvar_M_sup_S_drill_up) = (elit_Off));
        IF b1 THEN
            progress := TRUE;
            state1 := state0;

            state1.dvar_M_sup_S_drill_up := elit_On;

            state0 := state1;
        END_IF;
    END_IF;

    // Event "S_elevator_down_u_off".
    IF NOT progress THEN
        b1 := (state0.dvar_M_BoolToEventsTB) = (elit_X);
        b1 := b1 AND (NOT(ivar_s_elevator_down));
        b1 := b1 AND ((state0.dvar_M_sup_S_elevator_down) = (elit_On));
        IF b1 THEN
            progress := TRUE;
            state1 := state0;

            state1.dvar_M_sup_S_elevator_down := elit_Off;

            state0 := state1;
        END_IF;
    END_IF;

    // Event "S_elevator_down_u_on".
    IF NOT progress THEN
        b1 := (state0.dvar_M_BoolToEventsTB) = (elit_X);
        b1 := b1 AND (ivar_s_elevator_down);
        b1 := b1 AND ((state0.dvar_M_sup_S_elevator_down) = (elit_Off));
        b1 := b1 AND ((state0.dvar_M_sup_TDynamics) = (elit_X));
        b1 := b1 AND ((state0.dvar_M_sup_S_elevator_up) = (elit_Off));
        IF b1 THEN
            progress := TRUE;
            state1 := state0;

            state1.dvar_M_sup_S_elevator_down := elit_On;

            state0 := state1;
        END_IF;
    END_IF;

    // Event "S_elevator_up_u_off".
    IF NOT progress THEN
        b1 := (state0.dvar_M_BoolToEventsTB) = (elit_X);
        b1 := b1 AND (NOT(ivar_s_elevator_up));
        b1 := b1 AND ((state0.dvar_M_sup_S_elevator_up) = (elit_On));
        IF b1 THEN
            progress := TRUE;
            state1 := state0;

            state1.dvar_M_sup_S_elevator_up := elit_Off;

            state0 := state1;
        END_IF;
    END_IF;

    // Event "S_elevator_up_u_on".
    IF NOT progress THEN
        b1 := (state0.dvar_M_BoolToEventsTB) = (elit_X);
        b1 := b1 AND (ivar_s_elevator_up);
        b1 := b1 AND ((state0.dvar_M_sup_S_elevator_up) = (elit_Off));
        b1 := b1 AND ((state0.dvar_M_sup_TDynamics) = (elit_X));
        b1 := b1 AND ((state0.dvar_M_sup_S_elevator_down) = (elit_Off));
        IF b1 THEN
            progress := TRUE;
            state1 := state0;

            state1.dvar_M_sup_S_elevator_up := elit_On;

            state0 := state1;
        END_IF;
    END_IF;

    // Event "S_gate1_closed_u_off".
    IF NOT progress THEN
        b1 := (state0.dvar_M_BoolToEventsS) = (elit_X);
        b1 := b1 AND (NOT(ivar_s_gate1_closed));
        b1 := b1 AND ((state0.dvar_M_sup_S_gate1_closed) = (elit_On));
        IF b1 THEN
            progress := TRUE;
            state1 := state0;

            state1.dvar_M_sup_S_gate1_closed := elit_Off;

            state0 := state1;
        END_IF;
    END_IF;

    // Event "S_gate1_closed_u_on".
    IF NOT progress THEN
        b1 := (state0.dvar_M_BoolToEventsS) = (elit_X);
        b1 := b1 AND (ivar_s_gate1_closed);
        b1 := b1 AND ((state0.dvar_M_sup_S_gate1_closed) = (elit_Off));
        b1 := b1 AND ((state0.dvar_M_sup_SDynamics1) = (elit_X));
        b1 := b1 AND ((state0.dvar_M_sup_S_gate1_opened) = (elit_Off));
        IF b1 THEN
            progress := TRUE;
            state1 := state0;

            state1.dvar_M_sup_S_gate1_closed := elit_On;

            state0 := state1;
        END_IF;
    END_IF;

    // Event "S_gate1_opened_u_off".
    IF NOT progress THEN
        b1 := (state0.dvar_M_BoolToEventsS) = (elit_X);
        b1 := b1 AND (NOT(ivar_s_gate1_opened));
        b1 := b1 AND ((state0.dvar_M_sup_S_gate1_opened) = (elit_On));
        IF b1 THEN
            progress := TRUE;
            state1 := state0;

            state1.dvar_M_sup_S_gate1_opened := elit_Off;

            state0 := state1;
        END_IF;
    END_IF;

    // Event "S_gate1_opened_u_on".
    IF NOT progress THEN
        b1 := (state0.dvar_M_BoolToEventsS) = (elit_X);
        b1 := b1 AND (ivar_s_gate1_opened);
        b1 := b1 AND ((state0.dvar_M_sup_S_gate1_opened) = (elit_Off));
        b1 := b1 AND ((state0.dvar_M_sup_SDynamics1) = (elit_X));
        b1 := b1 AND ((state0.dvar_M_sup_S_gate1_closed) = (elit_Off));
        IF b1 THEN
            progress := TRUE;
            state1 := state0;

            state1.dvar_M_sup_S_gate1_opened := elit_On;

            state0 := state1;
        END_IF;
    END_IF;

    // Event "S_gate2_closed_u_off".
    IF NOT progress THEN
        b1 := (state0.dvar_M_BoolToEventsS) = (elit_X);
        b1 := b1 AND (NOT(ivar_s_gate2_closed));
        b1 := b1 AND ((state0.dvar_M_sup_S_gate2_closed) = (elit_On));
        IF b1 THEN
            progress := TRUE;
            state1 := state0;

            state1.dvar_M_sup_S_gate2_closed := elit_Off;

            state0 := state1;
        END_IF;
    END_IF;

    // Event "S_gate2_closed_u_on".
    IF NOT progress THEN
        b1 := (state0.dvar_M_BoolToEventsS) = (elit_X);
        b1 := b1 AND (ivar_s_gate2_closed);
        b1 := b1 AND ((state0.dvar_M_sup_S_gate2_closed) = (elit_Off));
        b1 := b1 AND ((state0.dvar_M_sup_SDynamics2) = (elit_X));
        b1 := b1 AND ((state0.dvar_M_sup_S_gate2_opened) = (elit_Off));
        IF b1 THEN
            progress := TRUE;
            state1 := state0;

            state1.dvar_M_sup_S_gate2_closed := elit_On;

            state0 := state1;
        END_IF;
    END_IF;

    // Event "S_gate2_opened_u_off".
    IF NOT progress THEN
        b1 := (state0.dvar_M_BoolToEventsS) = (elit_X);
        b1 := b1 AND (NOT(ivar_s_gate2_opened));
        b1 := b1 AND ((state0.dvar_M_sup_S_gate2_opened) = (elit_On));
        IF b1 THEN
            progress := TRUE;
            state1 := state0;

            state1.dvar_M_sup_S_gate2_opened := elit_Off;

            state0 := state1;
        END_IF;
    END_IF;

    // Event "S_gate2_opened_u_on".
    IF NOT progress THEN
        b1 := (state0.dvar_M_BoolToEventsS) = (elit_X);
        b1 := b1 AND (ivar_s_gate2_opened);
        b1 := b1 AND ((state0.dvar_M_sup_S_gate2_opened) = (elit_Off));
        b1 := b1 AND ((state0.dvar_M_sup_SDynamics2) = (elit_X));
        b1 := b1 AND ((state0.dvar_M_sup_S_gate2_closed) = (elit_Off));
        IF b1 THEN
            progress := TRUE;
            state1 := state0;

            state1.dvar_M_sup_S_gate2_opened := elit_On;

            state0 := state1;
        END_IF;
    END_IF;

    // Event "S_gripper_u_off".
    IF NOT progress THEN
        b1 := (state0.dvar_M_BoolToEventsDH) = (elit_X);
        b1 := b1 AND (NOT(ivar_s_gripper));
        b1 := b1 AND ((state0.dvar_M_sup_S_gripper) = (elit_On));
        IF b1 THEN
            progress := TRUE;
            state1 := state0;

            state1.dvar_M_sup_S_gripper := elit_Off;

            state0 := state1;
        END_IF;
    END_IF;

    // Event "S_gripper_u_on".
    IF NOT progress THEN
        b1 := (state0.dvar_M_BoolToEventsDH) = (elit_X);
        b1 := b1 AND (ivar_s_gripper);
        b1 := b1 AND ((state0.dvar_M_sup_S_gripper) = (elit_Off));
        IF b1 THEN
            progress := TRUE;
            state1 := state0;

            state1.dvar_M_sup_S_gripper := elit_On;

            state0 := state1;
        END_IF;
    END_IF;

    // Event "S_handlingbusy_u_off".
    IF NOT progress THEN
        b1 := (state0.dvar_M_BoolToEventsDH) = (elit_X);
        b1 := b1 AND (NOT(ivar_s_handlingbusy));
        b1 := b1 AND ((state0.dvar_M_sup_S_handlingbusy) = (elit_On));
        IF b1 THEN
            progress := TRUE;
            state1 := state0;

            state1.dvar_M_sup_S_handlingbusy := elit_Off;

            state0 := state1;
        END_IF;
    END_IF;

    // Event "S_handlingbusy_u_on".
    IF NOT progress THEN
        b1 := (state0.dvar_M_BoolToEventsDH) = (elit_X);
        b1 := b1 AND (ivar_s_handlingbusy);
        b1 := b1 AND ((state0.dvar_M_sup_S_handlingbusy) = (elit_Off));
        IF b1 THEN
            progress := TRUE;
            state1 := state0;

            state1.dvar_M_sup_S_handlingbusy := elit_On;

            state0 := state1;
        END_IF;
    END_IF;

    // Event "S_Hinitialized_u_off".
    IF NOT progress THEN
        b1 := (state0.dvar_M_BoolToEventsDH) = (elit_X);
        b1 := b1 AND ((state0.dvar_M_HardwareMapDH) <> (elit_initialized));
        b1 := b1 AND ((state0.dvar_M_sup_S_Hinitialized) = (elit_On));
        IF b1 THEN
            progress := TRUE;
            state1 := state0;

            state1.dvar_M_sup_S_Hinitialized := elit_Off;

            state0 := state1;
        END_IF;
    END_IF;

    // Event "S_Hinitialized_u_on".
    IF NOT progress THEN
        b1 := (state0.dvar_M_BoolToEventsDH) = (elit_X);
        b1 := b1 AND ((state0.dvar_M_HardwareMapDH) = (elit_initialized));
        b1 := b1 AND ((state0.dvar_M_sup_S_Hinitialized) = (elit_Off));
        IF b1 THEN
            progress := TRUE;
            state1 := state0;

            state1.dvar_M_sup_S_Hinitialized := elit_On;

            state0 := state1;
        END_IF;
    END_IF;

    // Event "S_inductive_u_off".
    IF NOT progress THEN
        b1 := (state0.dvar_M_BoolToEventsS) = (elit_X);
        b1 := b1 AND (NOT(ivar_s_inductive));
        b1 := b1 AND ((state0.dvar_M_sup_S_inductive) = (elit_On));
        IF b1 THEN
            progress := TRUE;
            state1 := state0;

            state1.dvar_M_sup_S_inductive := elit_Off;

            state0 := state1;
        END_IF;
    END_IF;

    // Event "S_inductive_u_on".
    IF NOT progress THEN
        b1 := (state0.dvar_M_BoolToEventsS) = (elit_X);
        b1 := b1 AND (ivar_s_inductive);
        b1 := b1 AND ((state0.dvar_M_sup_S_inductive) = (elit_Off));
        IF b1 THEN
            progress := TRUE;
            state1 := state0;

            state1.dvar_M_sup_S_inductive := elit_On;

            state0 := state1;
        END_IF;
    END_IF;

    // Event "S_optical_u_off".
    IF NOT progress THEN
        b1 := (state0.dvar_M_BoolToEventsS) = (elit_X);
        b1 := b1 AND (NOT(ivar_s_optical));
        b1 := b1 AND ((state0.dvar_M_sup_S_optical) = (elit_On));
        IF b1 THEN
            progress := TRUE;
            state1 := state0;

            state1.dvar_M_sup_S_optical := elit_Off;

            state0 := state1;
        END_IF;
    END_IF;

    // Event "S_optical_u_on".
    IF NOT progress THEN
        b1 := (state0.dvar_M_BoolToEventsS) = (elit_X);
        b1 := b1 AND (ivar_s_optical);
        b1 := b1 AND ((state0.dvar_M_sup_S_optical) = (elit_Off));
        IF b1 THEN
            progress := TRUE;
            state1 := state0;

            state1.dvar_M_sup_S_optical := elit_On;

            state0 := state1;
        END_IF;
    END_IF;

    // Event "S_opticalT_u_off".
    IF NOT progress THEN
        b1 := (state0.dvar_M_BoolToEventsTB) = (elit_X);
        b1 := b1 AND (NOT(ivar_s_opticalT));
        b1 := b1 AND ((state0.dvar_M_sup_S_opticalT) = (elit_On));
        IF b1 THEN
            progress := TRUE;
            state1 := state0;

            state1.dvar_M_sup_S_opticalT := elit_Off;

            state0 := state1;
        END_IF;
    END_IF;

    // Event "S_opticalT_u_on".
    IF NOT progress THEN
        b1 := (state0.dvar_M_BoolToEventsTB) = (elit_X);
        b1 := b1 AND (ivar_s_opticalT);
        b1 := b1 AND ((state0.dvar_M_sup_S_opticalT) = (elit_Off));
        IF b1 THEN
            progress := TRUE;
            state1 := state0;

            state1.dvar_M_sup_S_opticalT := elit_On;

            state0 := state1;
        END_IF;
    END_IF;

    // Event "S_Pinitialized_u_off".
    IF NOT progress THEN
        b1 := (state0.dvar_M_BoolToEventsP) = (elit_X);
        b1 := b1 AND ((state0.dvar_M_HardwareMapP) <> (elit_initialized));
        b1 := b1 AND ((state0.dvar_M_sup_S_Pinitialized) = (elit_On));
        IF b1 THEN
            progress := TRUE;
            state1 := state0;

            state1.dvar_M_sup_S_Pinitialized := elit_Off;

            state0 := state1;
        END_IF;
    END_IF;

    // Event "S_Pinitialized_u_on".
    IF NOT progress THEN
        b1 := (state0.dvar_M_BoolToEventsP) = (elit_X);
        b1 := b1 AND ((state0.dvar_M_HardwareMapP) = (elit_initialized));
        b1 := b1 AND ((state0.dvar_M_sup_S_Pinitialized) = (elit_Off));
        IF b1 THEN
            progress := TRUE;
            state1 := state0;

            state1.dvar_M_sup_S_Pinitialized := elit_On;

            state0 := state1;
        END_IF;
    END_IF;

    // Event "S_processingbusy_u_off".
    IF NOT progress THEN
        b1 := (state0.dvar_M_BoolToEventsTB) = (elit_X);
        b1 := b1 AND (NOT(ivar_s_processingbusy));
        b1 := b1 AND ((state0.dvar_M_sup_S_processingbusy) = (elit_On));
        IF b1 THEN
            progress := TRUE;
            state1 := state0;

            state1.dvar_M_sup_S_processingbusy := elit_Off;

            state0 := state1;
        END_IF;
    END_IF;

    // Event "S_processingbusy_u_on".
    IF NOT progress THEN
        b1 := (state0.dvar_M_BoolToEventsTB) = (elit_X);
        b1 := b1 AND (ivar_s_processingbusy);
        b1 := b1 AND ((state0.dvar_M_sup_S_processingbusy) = (elit_Off));
        IF b1 THEN
            progress := TRUE;
            state1 := state0;

            state1.dvar_M_sup_S_processingbusy := elit_On;

            state0 := state1;
        END_IF;
    END_IF;

    // Event "S_product_u_off".
    IF NOT progress THEN
        b1 := (state0.dvar_M_BoolToEventsS) = (elit_X);
        b1 := b1 AND (NOT(ivar_s_product));
        b1 := b1 AND ((state0.dvar_M_sup_S_product) = (elit_On));
        IF b1 THEN
            progress := TRUE;
            state1 := state0;

            state1.dvar_M_sup_S_product := elit_Off;

            state0 := state1;
        END_IF;
    END_IF;

    // Event "S_product_u_on".
    IF NOT progress THEN
        b1 := (state0.dvar_M_BoolToEventsS) = (elit_X);
        b1 := b1 AND (ivar_s_product);
        b1 := b1 AND ((state0.dvar_M_sup_S_product) = (elit_Off));
        IF b1 THEN
            progress := TRUE;
            state1 := state0;

            state1.dvar_M_sup_S_product := elit_On;

            state0 := state1;
        END_IF;
    END_IF;

    // Event "S_product1_u_off".
    IF NOT progress THEN
        b1 := (state0.dvar_M_BoolToEventsDH) = (elit_X);
        IF b1 THEN
            b2 := NOT(ivar_s_product1);
            b2 := b2 OR (NOT(ivar_s_product1));
            b1 := b1 AND (b2);
        END_IF;
        b1 := b1 AND ((state0.dvar_M_sup_S_product1) = (elit_On));
        IF b1 THEN
            progress := TRUE;
            state1 := state0;

            state1.dvar_M_sup_S_product1 := elit_Off;

            state0 := state1;
        END_IF;
    END_IF;

    // Event "S_product1_u_on".
    IF NOT progress THEN
        b1 := (state0.dvar_M_BoolToEventsDH) = (elit_X);
        IF b1 THEN
            b2 := ivar_s_product1;
            b2 := b2 OR (ivar_s_product1);
            b1 := b1 AND (b2);
        END_IF;
        b1 := b1 AND ((state0.dvar_M_sup_S_product1) = (elit_Off));
        IF b1 THEN
            progress := TRUE;
            state1 := state0;

            state1.dvar_M_sup_S_product1 := elit_On;

            state0 := state1;
        END_IF;
    END_IF;

    // Event "S_product2_u_off".
    IF NOT progress THEN
        b1 := (state0.dvar_M_BoolToEventsDH) = (elit_X);
        IF b1 THEN
            b2 := NOT(ivar_s_product2);
            b2 := b2 OR (NOT(ivar_s_product2));
            b1 := b1 AND (b2);
        END_IF;
        b1 := b1 AND ((state0.dvar_M_sup_S_product2) = (elit_On));
        IF b1 THEN
            progress := TRUE;
            state1 := state0;

            state1.dvar_M_sup_S_product2 := elit_Off;

            state0 := state1;
        END_IF;
    END_IF;

    // Event "S_product2_u_on".
    IF NOT progress THEN
        b1 := (state0.dvar_M_BoolToEventsDH) = (elit_X);
        IF b1 THEN
            b2 := ivar_s_product2;
            b2 := b2 OR (ivar_s_product2);
            b1 := b1 AND (b2);
        END_IF;
        b1 := b1 AND ((state0.dvar_M_sup_S_product2) = (elit_Off));
        IF b1 THEN
            progress := TRUE;
            state1 := state0;

            state1.dvar_M_sup_S_product2 := elit_On;

            state0 := state1;
        END_IF;
    END_IF;

    // Event "S_product3_u_off".
    IF NOT progress THEN
        b1 := (state0.dvar_M_BoolToEventsDH) = (elit_X);
        IF b1 THEN
            b2 := NOT(ivar_s_product3);
            b2 := b2 OR (NOT(ivar_s_product3));
            b1 := b1 AND (b2);
        END_IF;
        b1 := b1 AND ((state0.dvar_M_sup_S_product3) = (elit_On));
        IF b1 THEN
            progress := TRUE;
            state1 := state0;

            state1.dvar_M_sup_S_product3 := elit_Off;

            state0 := state1;
        END_IF;
    END_IF;

    // Event "S_product3_u_on".
    IF NOT progress THEN
        b1 := (state0.dvar_M_BoolToEventsDH) = (elit_X);
        IF b1 THEN
            b2 := ivar_s_product3;
            b2 := b2 OR (ivar_s_product3);
            b1 := b1 AND (b2);
        END_IF;
        b1 := b1 AND ((state0.dvar_M_sup_S_product3) = (elit_Off));
        IF b1 THEN
            progress := TRUE;
            state1 := state0;

            state1.dvar_M_sup_S_product3 := elit_On;

            state0 := state1;
        END_IF;
    END_IF;

    // Event "S_product4_u_off".
    IF NOT progress THEN
        b1 := (state0.dvar_M_BoolToEventsDH) = (elit_X);
        b1 := b1 AND (NOT(ivar_s_product4));
        b1 := b1 AND ((state0.dvar_M_sup_S_product4) = (elit_On));
        IF b1 THEN
            progress := TRUE;
            state1 := state0;

            state1.dvar_M_sup_S_product4 := elit_Off;

            state0 := state1;
        END_IF;
    END_IF;

    // Event "S_product4_u_on".
    IF NOT progress THEN
        b1 := (state0.dvar_M_BoolToEventsDH) = (elit_X);
        b1 := b1 AND (ivar_s_product4);
        b1 := b1 AND ((state0.dvar_M_sup_S_product4) = (elit_Off));
        IF b1 THEN
            progress := TRUE;
            state1 := state0;

            state1.dvar_M_sup_S_product4 := elit_On;

            state0 := state1;
        END_IF;
    END_IF;

    // Event "S_productheight_u_off".
    IF NOT progress THEN
        b1 := (state0.dvar_M_BoolToEventsTB) = (elit_X);
        b1 := b1 AND (NOT(ivar_s_productheight));
        b1 := b1 AND ((state0.dvar_M_sup_S_productheight) = (elit_On));
        IF b1 THEN
            progress := TRUE;
            state1 := state0;

            state1.dvar_M_sup_S_productheight := elit_Off;

            state0 := state1;
        END_IF;
    END_IF;

    // Event "S_productheight_u_on".
    IF NOT progress THEN
        b1 := (state0.dvar_M_BoolToEventsTB) = (elit_X);
        b1 := b1 AND (ivar_s_productheight);
        b1 := b1 AND ((state0.dvar_M_sup_S_productheight) = (elit_Off));
        IF b1 THEN
            progress := TRUE;
            state1 := state0;

            state1.dvar_M_sup_S_productheight := elit_On;

            state0 := state1;
        END_IF;
    END_IF;

    // Event "S_pusher_u_off".
    IF NOT progress THEN
        b1 := (state0.dvar_M_BoolToEventsTB) = (elit_X);
        b1 := b1 AND (NOT(ivar_s_pusher));
        b1 := b1 AND ((state0.dvar_M_sup_S_pusher) = (elit_On));
        IF b1 THEN
            progress := TRUE;
            state1 := state0;

            state1.dvar_M_sup_S_pusher := elit_Off;

            state0 := state1;
        END_IF;
    END_IF;

    // Event "S_pusher_u_on".
    IF NOT progress THEN
        b1 := (state0.dvar_M_BoolToEventsTB) = (elit_X);
        b1 := b1 AND (ivar_s_pusher);
        b1 := b1 AND ((state0.dvar_M_sup_S_pusher) = (elit_Off));
        IF b1 THEN
            progress := TRUE;
            state1 := state0;

            state1.dvar_M_sup_S_pusher := elit_On;

            state0 := state1;
        END_IF;
    END_IF;

    // Event "S_pusher1_in_u_off".
    IF NOT progress THEN
        b1 := (state0.dvar_M_BoolToEventsDH) = (elit_X);
        b1 := b1 AND (NOT(ivar_s_pusher1_in));
        b1 := b1 AND ((state0.dvar_M_sup_S_pusher1_in) = (elit_On));
        IF b1 THEN
            progress := TRUE;
            state1 := state0;

            state1.dvar_M_sup_S_pusher1_in := elit_Off;

            state0 := state1;
        END_IF;
    END_IF;

    // Event "S_pusher1_in_u_on".
    IF NOT progress THEN
        b1 := (state0.dvar_M_BoolToEventsDH) = (elit_X);
        b1 := b1 AND (ivar_s_pusher1_in);
        b1 := b1 AND ((state0.dvar_M_sup_DDynamics1) = (elit_X));
        b1 := b1 AND ((state0.dvar_M_sup_S_pusher1_out) = (elit_Off));
        b1 := b1 AND ((state0.dvar_M_sup_S_pusher1_in) = (elit_Off));
        IF b1 THEN
            progress := TRUE;
            state1 := state0;

            state1.dvar_M_sup_S_pusher1_in := elit_On;

            state0 := state1;
        END_IF;
    END_IF;

    // Event "S_pusher1_out_u_off".
    IF NOT progress THEN
        b1 := (state0.dvar_M_BoolToEventsDH) = (elit_X);
        b1 := b1 AND (NOT(ivar_s_pusher1_out));
        b1 := b1 AND ((state0.dvar_M_sup_S_pusher1_out) = (elit_On));
        IF b1 THEN
            progress := TRUE;
            state1 := state0;

            state1.dvar_M_sup_S_pusher1_out := elit_Off;

            state0 := state1;
        END_IF;
    END_IF;

    // Event "S_pusher1_out_u_on".
    IF NOT progress THEN
        b1 := (state0.dvar_M_BoolToEventsDH) = (elit_X);
        b1 := b1 AND (ivar_s_pusher1_out);
        b1 := b1 AND ((state0.dvar_M_sup_DDynamics1) = (elit_X));
        b1 := b1 AND ((state0.dvar_M_sup_S_pusher1_in) = (elit_Off));
        b1 := b1 AND ((state0.dvar_M_sup_S_pusher1_out) = (elit_Off));
        IF b1 THEN
            progress := TRUE;
            state1 := state0;

            state1.dvar_M_sup_S_pusher1_out := elit_On;

            state0 := state1;
        END_IF;
    END_IF;

    // Event "S_pusher2_in_u_off".
    IF NOT progress THEN
        b1 := (state0.dvar_M_BoolToEventsDH) = (elit_X);
        b1 := b1 AND (NOT(ivar_s_pusher2_in));
        b1 := b1 AND ((state0.dvar_M_sup_S_pusher2_in) = (elit_On));
        IF b1 THEN
            progress := TRUE;
            state1 := state0;

            state1.dvar_M_sup_S_pusher2_in := elit_Off;

            state0 := state1;
        END_IF;
    END_IF;

    // Event "S_pusher2_in_u_on".
    IF NOT progress THEN
        b1 := (state0.dvar_M_BoolToEventsDH) = (elit_X);
        b1 := b1 AND (ivar_s_pusher2_in);
        b1 := b1 AND ((state0.dvar_M_sup_DDynamics2) = (elit_X));
        b1 := b1 AND ((state0.dvar_M_sup_S_pusher2_out) = (elit_Off));
        b1 := b1 AND ((state0.dvar_M_sup_S_pusher2_in) = (elit_Off));
        IF b1 THEN
            progress := TRUE;
            state1 := state0;

            state1.dvar_M_sup_S_pusher2_in := elit_On;

            state0 := state1;
        END_IF;
    END_IF;

    // Event "S_pusher2_out_u_off".
    IF NOT progress THEN
        b1 := (state0.dvar_M_BoolToEventsDH) = (elit_X);
        b1 := b1 AND (NOT(ivar_s_pusher2_out));
        b1 := b1 AND ((state0.dvar_M_sup_S_pusher2_out) = (elit_On));
        IF b1 THEN
            progress := TRUE;
            state1 := state0;

            state1.dvar_M_sup_S_pusher2_out := elit_Off;

            state0 := state1;
        END_IF;
    END_IF;

    // Event "S_pusher2_out_u_on".
    IF NOT progress THEN
        b1 := (state0.dvar_M_BoolToEventsDH) = (elit_X);
        b1 := b1 AND (ivar_s_pusher2_out);
        b1 := b1 AND ((state0.dvar_M_sup_DDynamics2) = (elit_X));
        b1 := b1 AND ((state0.dvar_M_sup_S_pusher2_in) = (elit_Off));
        b1 := b1 AND ((state0.dvar_M_sup_S_pusher2_out) = (elit_Off));
        IF b1 THEN
            progress := TRUE;
            state1 := state0;

            state1.dvar_M_sup_S_pusher2_out := elit_On;

            state0 := state1;
        END_IF;
    END_IF;

    // Event "S_pusher3_in_u_off".
    IF NOT progress THEN
        b1 := (state0.dvar_M_BoolToEventsDH) = (elit_X);
        b1 := b1 AND (NOT(ivar_s_pusher3_in));
        b1 := b1 AND ((state0.dvar_M_sup_S_pusher3_in) = (elit_On));
        IF b1 THEN
            progress := TRUE;
            state1 := state0;

            state1.dvar_M_sup_S_pusher3_in := elit_Off;

            state0 := state1;
        END_IF;
    END_IF;

    // Event "S_pusher3_in_u_on".
    IF NOT progress THEN
        b1 := (state0.dvar_M_BoolToEventsDH) = (elit_X);
        b1 := b1 AND (ivar_s_pusher3_in);
        b1 := b1 AND ((state0.dvar_M_sup_DDynamics3) = (elit_X));
        b1 := b1 AND ((state0.dvar_M_sup_S_pusher3_out) = (elit_Off));
        b1 := b1 AND ((state0.dvar_M_sup_S_pusher3_in) = (elit_Off));
        IF b1 THEN
            progress := TRUE;
            state1 := state0;

            state1.dvar_M_sup_S_pusher3_in := elit_On;

            state0 := state1;
        END_IF;
    END_IF;

    // Event "S_pusher3_out_u_off".
    IF NOT progress THEN
        b1 := (state0.dvar_M_BoolToEventsDH) = (elit_X);
        b1 := b1 AND (NOT(ivar_s_pusher3_out));
        b1 := b1 AND ((state0.dvar_M_sup_S_pusher3_out) = (elit_On));
        IF b1 THEN
            progress := TRUE;
            state1 := state0;

            state1.dvar_M_sup_S_pusher3_out := elit_Off;

            state0 := state1;
        END_IF;
    END_IF;

    // Event "S_pusher3_out_u_on".
    IF NOT progress THEN
        b1 := (state0.dvar_M_BoolToEventsDH) = (elit_X);
        b1 := b1 AND (ivar_s_pusher3_out);
        b1 := b1 AND ((state0.dvar_M_sup_DDynamics3) = (elit_X));
        b1 := b1 AND ((state0.dvar_M_sup_S_pusher3_in) = (elit_Off));
        b1 := b1 AND ((state0.dvar_M_sup_S_pusher3_out) = (elit_Off));
        IF b1 THEN
            progress := TRUE;
            state1 := state0;

            state1.dvar_M_sup_S_pusher3_out := elit_On;

            state0 := state1;
        END_IF;
    END_IF;

    // Event "S_reflective_u_off".
    IF NOT progress THEN
        b1 := (state0.dvar_M_BoolToEventsTB) = (elit_X);
        b1 := b1 AND (NOT(ivar_s_reflective));
        b1 := b1 AND ((state0.dvar_M_sup_S_reflective) = (elit_On));
        IF b1 THEN
            progress := TRUE;
            state1 := state0;

            state1.dvar_M_sup_S_reflective := elit_Off;

            state0 := state1;
        END_IF;
    END_IF;

    // Event "S_reflective_u_on".
    IF NOT progress THEN
        b1 := (state0.dvar_M_BoolToEventsTB) = (elit_X);
        b1 := b1 AND (ivar_s_reflective);
        b1 := b1 AND ((state0.dvar_M_sup_S_reflective) = (elit_Off));
        IF b1 THEN
            progress := TRUE;
            state1 := state0;

            state1.dvar_M_sup_S_reflective := elit_On;

            state0 := state1;
        END_IF;
    END_IF;

    // Event "S_separator_closed_u_off".
    IF NOT progress THEN
        b1 := (state0.dvar_M_BoolToEventsTB) = (elit_X);
        b1 := b1 AND (NOT(ivar_s_separator_closed));
        b1 := b1 AND ((state0.dvar_M_sup_S_separator_closed) = (elit_On));
        IF b1 THEN
            progress := TRUE;
            state1 := state0;

            state1.dvar_M_sup_S_separator_closed := elit_Off;

            state0 := state1;
        END_IF;
    END_IF;

    // Event "S_separator_closed_u_on".
    IF NOT progress THEN
        b1 := (state0.dvar_M_BoolToEventsTB) = (elit_X);
        b1 := b1 AND (ivar_s_separator_closed);
        b1 := b1 AND ((state0.dvar_M_sup_BDynamics) = (elit_X));
        b1 := b1 AND ((state0.dvar_M_sup_S_separator_opened) = (elit_Off));
        b1 := b1 AND ((state0.dvar_M_sup_S_separator_closed) = (elit_Off));
        IF b1 THEN
            progress := TRUE;
            state1 := state0;

            state1.dvar_M_sup_S_separator_closed := elit_On;

            state0 := state1;
        END_IF;
    END_IF;

    // Event "S_separator_opened_u_off".
    IF NOT progress THEN
        b1 := (state0.dvar_M_BoolToEventsTB) = (elit_X);
        b1 := b1 AND (NOT(ivar_s_separator_opened));
        b1 := b1 AND ((state0.dvar_M_sup_S_separator_opened) = (elit_On));
        IF b1 THEN
            progress := TRUE;
            state1 := state0;

            state1.dvar_M_sup_S_separator_opened := elit_Off;

            state0 := state1;
        END_IF;
    END_IF;

    // Event "S_separator_opened_u_on".
    IF NOT progress THEN
        b1 := (state0.dvar_M_BoolToEventsTB) = (elit_X);
        b1 := b1 AND (ivar_s_separator_opened);
        b1 := b1 AND ((state0.dvar_M_sup_BDynamics) = (elit_X));
        b1 := b1 AND ((state0.dvar_M_sup_S_separator_closed) = (elit_Off));
        b1 := b1 AND ((state0.dvar_M_sup_S_separator_opened) = (elit_Off));
        IF b1 THEN
            progress := TRUE;
            state1 := state0;

            state1.dvar_M_sup_S_separator_opened := elit_On;

            state0 := state1;
        END_IF;
    END_IF;

    // Event "S_Sinitialized_u_off".
    IF NOT progress THEN
        b1 := (state0.dvar_M_BoolToEventsS) = (elit_X);
        b1 := b1 AND ((state0.dvar_M_HardwareMapS) <> (elit_initialized));
        b1 := b1 AND ((state0.dvar_M_sup_S_Sinitialized) = (elit_On));
        IF b1 THEN
            progress := TRUE;
            state1 := state0;

            state1.dvar_M_sup_S_Sinitialized := elit_Off;

            state0 := state1;
        END_IF;
    END_IF;

    // Event "S_Sinitialized_u_on".
    IF NOT progress THEN
        b1 := (state0.dvar_M_BoolToEventsS) = (elit_X);
        b1 := b1 AND ((state0.dvar_M_HardwareMapS) = (elit_initialized));
        b1 := b1 AND ((state0.dvar_M_sup_S_Sinitialized) = (elit_Off));
        IF b1 THEN
            progress := TRUE;
            state1 := state0;

            state1.dvar_M_sup_S_Sinitialized := elit_On;

            state0 := state1;
        END_IF;
    END_IF;

    // Event "S_slidefull_u_off".
    IF NOT progress THEN
        b1 := (state0.dvar_M_BoolToEventsS) = (elit_X);
        b1 := b1 AND (NOT(ivar_s_slidefull));
        b1 := b1 AND ((state0.dvar_M_sup_S_slidefull) = (elit_On));
        IF b1 THEN
            progress := TRUE;
            state1 := state0;

            state1.dvar_M_sup_S_slidefull := elit_Off;

            state0 := state1;
        END_IF;
    END_IF;

    // Event "S_slidefull_u_on".
    IF NOT progress THEN
        b1 := (state0.dvar_M_BoolToEventsS) = (elit_X);
        b1 := b1 AND (ivar_s_slidefull);
        b1 := b1 AND ((state0.dvar_M_sup_S_slidefull) = (elit_Off));
        IF b1 THEN
            progress := TRUE;
            state1 := state0;

            state1.dvar_M_sup_S_slidefull := elit_On;

            state0 := state1;
        END_IF;
    END_IF;

    // Event "S_sortingbusy_u_off".
    IF NOT progress THEN
        b1 := (state0.dvar_M_BoolToEventsP) = (elit_X);
        b1 := b1 AND (NOT(ivar_s_sortingbusy));
        b1 := b1 AND ((state0.dvar_M_sup_S_sortingbusy) = (elit_On));
        IF b1 THEN
            progress := TRUE;
            state1 := state0;

            state1.dvar_M_sup_S_sortingbusy := elit_Off;

            state0 := state1;
        END_IF;
    END_IF;

    // Event "S_sortingbusy_u_on".
    IF NOT progress THEN
        b1 := (state0.dvar_M_BoolToEventsP) = (elit_X);
        b1 := b1 AND (ivar_s_sortingbusy);
        b1 := b1 AND ((state0.dvar_M_sup_S_sortingbusy) = (elit_Off));
        IF b1 THEN
            progress := TRUE;
            state1 := state0;

            state1.dvar_M_sup_S_sortingbusy := elit_On;

            state0 := state1;
        END_IF;
    END_IF;

    // Event "S_stack1_filled_u_off".
    IF NOT progress THEN
        b1 := (state0.dvar_M_BoolToEventsDH) = (elit_X);
        b1 := b1 AND (NOT(ivar_s_stack1filled));
        b1 := b1 AND ((state0.dvar_M_sup_S_stack1_filled) = (elit_On));
        IF b1 THEN
            progress := TRUE;
            state1 := state0;

            state1.dvar_M_sup_S_stack1_filled := elit_Off;

            state0 := state1;
        END_IF;
    END_IF;

    // Event "S_stack1_filled_u_on".
    IF NOT progress THEN
        b1 := (state0.dvar_M_BoolToEventsDH) = (elit_X);
        b1 := b1 AND (ivar_s_stack1filled);
        b1 := b1 AND ((state0.dvar_M_sup_S_stack1_filled) = (elit_Off));
        IF b1 THEN
            progress := TRUE;
            state1 := state0;

            state1.dvar_M_sup_S_stack1_filled := elit_On;

            state0 := state1;
        END_IF;
    END_IF;

    // Event "S_stack2_filled_u_off".
    IF NOT progress THEN
        b1 := (state0.dvar_M_BoolToEventsDH) = (elit_X);
        b1 := b1 AND (NOT(ivar_s_stack2filled));
        b1 := b1 AND ((state0.dvar_M_sup_S_stack2_filled) = (elit_On));
        IF b1 THEN
            progress := TRUE;
            state1 := state0;

            state1.dvar_M_sup_S_stack2_filled := elit_Off;

            state0 := state1;
        END_IF;
    END_IF;

    // Event "S_stack2_filled_u_on".
    IF NOT progress THEN
        b1 := (state0.dvar_M_BoolToEventsDH) = (elit_X);
        b1 := b1 AND (ivar_s_stack2filled);
        b1 := b1 AND ((state0.dvar_M_sup_S_stack2_filled) = (elit_Off));
        IF b1 THEN
            progress := TRUE;
            state1 := state0;

            state1.dvar_M_sup_S_stack2_filled := elit_On;

            state0 := state1;
        END_IF;
    END_IF;

    // Event "S_stack3_filled_u_off".
    IF NOT progress THEN
        b1 := (state0.dvar_M_BoolToEventsDH) = (elit_X);
        b1 := b1 AND (NOT(ivar_s_stack3filled));
        b1 := b1 AND ((state0.dvar_M_sup_S_stack3_filled) = (elit_On));
        IF b1 THEN
            progress := TRUE;
            state1 := state0;

            state1.dvar_M_sup_S_stack3_filled := elit_Off;

            state0 := state1;
        END_IF;
    END_IF;

    // Event "S_stack3_filled_u_on".
    IF NOT progress THEN
        b1 := (state0.dvar_M_BoolToEventsDH) = (elit_X);
        b1 := b1 AND (ivar_s_stack3filled);
        b1 := b1 AND ((state0.dvar_M_sup_S_stack3_filled) = (elit_Off));
        IF b1 THEN
            progress := TRUE;
            state1 := state0;

            state1.dvar_M_sup_S_stack3_filled := elit_On;

            state0 := state1;
        END_IF;
    END_IF;

    // Event "S_test_ok_u_off".
    IF NOT progress THEN
        b1 := (state0.dvar_M_BoolToEventsP) = (elit_X);
        b1 := b1 AND (NOT(ivar_s_test_ok));
        b1 := b1 AND ((state0.dvar_M_sup_S_test_ok) = (elit_On));
        IF b1 THEN
            progress := TRUE;
            state1 := state0;

            state1.dvar_M_sup_S_test_ok := elit_Off;

            state0 := state1;
        END_IF;
    END_IF;

    // Event "S_test_ok_u_on".
    IF NOT progress THEN
        b1 := (state0.dvar_M_BoolToEventsP) = (elit_X);
        b1 := b1 AND (ivar_s_test_ok);
        b1 := b1 AND ((state0.dvar_M_sup_S_test_ok) = (elit_Off));
        IF b1 THEN
            progress := TRUE;
            state1 := state0;

            state1.dvar_M_sup_S_test_ok := elit_On;

            state0 := state1;
        END_IF;
    END_IF;

    // Event "S_testingbusy_u_off".
    IF NOT progress THEN
        b1 := (state0.dvar_M_BoolToEventsDH) = (elit_X);
        b1 := b1 AND (NOT(ivar_s_testingbusy));
        b1 := b1 AND ((state0.dvar_M_sup_S_testingbusy) = (elit_On));
        IF b1 THEN
            progress := TRUE;
            state1 := state0;

            state1.dvar_M_sup_S_testingbusy := elit_Off;

            state0 := state1;
        END_IF;
    END_IF;

    // Event "S_testingbusy_u_on".
    IF NOT progress THEN
        b1 := (state0.dvar_M_BoolToEventsDH) = (elit_X);
        b1 := b1 AND (ivar_s_testingbusy);
        b1 := b1 AND ((state0.dvar_M_sup_S_testingbusy) = (elit_Off));
        IF b1 THEN
            progress := TRUE;
            state1 := state0;

            state1.dvar_M_sup_S_testingbusy := elit_On;

            state0 := state1;
        END_IF;
    END_IF;

    // Event "S_Tinitialized_u_off".
    IF NOT progress THEN
        b1 := (state0.dvar_M_BoolToEventsTB) = (elit_X);
        b1 := b1 AND ((state0.dvar_M_HardwareMapTB) <> (elit_initialized));
        b1 := b1 AND ((state0.dvar_M_sup_S_Tinitialized) = (elit_On));
        IF b1 THEN
            progress := TRUE;
            state1 := state0;

            state1.dvar_M_sup_S_Tinitialized := elit_Off;

            state0 := state1;
        END_IF;
    END_IF;

    // Event "S_Tinitialized_u_on".
    IF NOT progress THEN
        b1 := (state0.dvar_M_BoolToEventsTB) = (elit_X);
        b1 := b1 AND ((state0.dvar_M_HardwareMapTB) = (elit_initialized));
        b1 := b1 AND ((state0.dvar_M_sup_S_Tinitialized) = (elit_Off));
        IF b1 THEN
            progress := TRUE;
            state1 := state0;

            state1.dvar_M_sup_S_Tinitialized := elit_On;

            state0 := state1;
        END_IF;
    END_IF;

    // Event "S_transfer_atdrop_u_off".
    IF NOT progress THEN
        b1 := (state0.dvar_M_BoolToEventsDH) = (elit_X);
        b1 := b1 AND (NOT(ivar_s_transfer_atdrop));
        b1 := b1 AND ((state0.dvar_M_sup_S_transfer_atdrop) = (elit_On));
        IF b1 THEN
            progress := TRUE;
            state1 := state0;

            state1.dvar_M_sup_S_transfer_atdrop := elit_Off;

            state0 := state1;
        END_IF;
    END_IF;

    // Event "S_transfer_atdrop_u_on".
    IF NOT progress THEN
        b1 := (state0.dvar_M_BoolToEventsDH) = (elit_X);
        b1 := b1 AND (ivar_s_transfer_atdrop);
        b1 := b1 AND ((state0.dvar_M_sup_HDynamics2) = (elit_X));
        b1 := b1 AND ((state0.dvar_M_sup_S_transfer_atpickup) = (elit_Off));
        b1 := b1 AND ((state0.dvar_M_sup_S_transfer_athalfway) = (elit_Off));
        b1 := b1 AND ((state0.dvar_M_sup_S_transfer_atdrop) = (elit_Off));
        IF b1 THEN
            progress := TRUE;
            state1 := state0;

            state1.dvar_M_sup_S_transfer_atdrop := elit_On;

            state0 := state1;
        END_IF;
    END_IF;

    // Event "S_transfer_athalfway_u_off".
    IF NOT progress THEN
        b1 := (state0.dvar_M_BoolToEventsDH) = (elit_X);
        b1 := b1 AND (NOT(ivar_s_transfer_athalfway));
        b1 := b1 AND ((state0.dvar_M_sup_S_transfer_athalfway) = (elit_On));
        IF b1 THEN
            progress := TRUE;
            state1 := state0;

            state1.dvar_M_sup_S_transfer_athalfway := elit_Off;

            state0 := state1;
        END_IF;
    END_IF;

    // Event "S_transfer_athalfway_u_on".
    IF NOT progress THEN
        b1 := (state0.dvar_M_BoolToEventsDH) = (elit_X);
        b1 := b1 AND (ivar_s_transfer_athalfway);
        b1 := b1 AND ((state0.dvar_M_sup_HDynamics2) = (elit_X));
        b1 := b1 AND ((state0.dvar_M_sup_S_transfer_atdrop) = (elit_Off));
        b1 := b1 AND ((state0.dvar_M_sup_S_transfer_atpickup) = (elit_Off));
        b1 := b1 AND ((state0.dvar_M_sup_S_transfer_athalfway) = (elit_Off));
        IF b1 THEN
            progress := TRUE;
            state1 := state0;

            state1.dvar_M_sup_S_transfer_athalfway := elit_On;

            state0 := state1;
        END_IF;
    END_IF;

    // Event "S_transfer_atpickup_u_off".
    IF NOT progress THEN
        b1 := (state0.dvar_M_BoolToEventsDH) = (elit_X);
        b1 := b1 AND (NOT(ivar_s_transfer_atpickup));
        b1 := b1 AND ((state0.dvar_M_sup_S_transfer_atpickup) = (elit_On));
        IF b1 THEN
            progress := TRUE;
            state1 := state0;

            state1.dvar_M_sup_S_transfer_atpickup := elit_Off;

            state0 := state1;
        END_IF;
    END_IF;

    // Event "S_transfer_atpickup_u_on".
    IF NOT progress THEN
        b1 := (state0.dvar_M_BoolToEventsDH) = (elit_X);
        b1 := b1 AND (ivar_s_transfer_atpickup);
        b1 := b1 AND ((state0.dvar_M_sup_HDynamics2) = (elit_X));
        b1 := b1 AND ((state0.dvar_M_sup_S_transfer_atdrop) = (elit_Off));
        b1 := b1 AND ((state0.dvar_M_sup_S_transfer_athalfway) = (elit_Off));
        b1 := b1 AND ((state0.dvar_M_sup_S_transfer_atpickup) = (elit_Off));
        IF b1 THEN
            progress := TRUE;
            state1 := state0;

            state1.dvar_M_sup_S_transfer_atpickup := elit_On;

            state0 := state1;
        END_IF;
    END_IF;

    // Event "S_turntable_u_off".
    IF NOT progress THEN
        b1 := (state0.dvar_M_BoolToEventsP) = (elit_X);
        b1 := b1 AND (NOT(ivar_s_turntable));
        b1 := b1 AND ((state0.dvar_M_sup_S_turntable) = (elit_On));
        IF b1 THEN
            progress := TRUE;
            state1 := state0;

            state1.dvar_M_sup_S_turntable := elit_Off;

            state0 := state1;
        END_IF;
    END_IF;

    // Event "S_turntable_u_on".
    IF NOT progress THEN
        b1 := (state0.dvar_M_BoolToEventsP) = (elit_X);
        b1 := b1 AND (ivar_s_turntable);
        b1 := b1 AND ((state0.dvar_M_sup_S_turntable) = (elit_Off));
        IF b1 THEN
            progress := TRUE;
            state1 := state0;

            state1.dvar_M_sup_S_turntable := elit_On;

            state0 := state1;
        END_IF;
    END_IF;

    // Event "S_vacuum_u_off".
    IF NOT progress THEN
        b1 := (state0.dvar_M_BoolToEventsDH) = (elit_X);
        b1 := b1 AND (NOT(ivar_s_vacuum));
        b1 := b1 AND ((state0.dvar_M_sup_S_vacuum) = (elit_On));
        IF b1 THEN
            progress := TRUE;
            state1 := state0;

            state1.dvar_M_sup_S_vacuum := elit_Off;

            state0 := state1;
        END_IF;
    END_IF;

    // Event "S_vacuum_u_on".
    IF NOT progress THEN
        b1 := (state0.dvar_M_BoolToEventsDH) = (elit_X);
        b1 := b1 AND (ivar_s_vacuum);
        b1 := b1 AND ((state0.dvar_M_sup_S_vacuum) = (elit_Off));
        IF b1 THEN
            progress := TRUE;
            state1 := state0;

            state1.dvar_M_sup_S_vacuum := elit_On;

            state0 := state1;
        END_IF;
    END_IF;

    // Event "S_xpos_at1_u_off".
    IF NOT progress THEN
        b1 := (state0.dvar_M_BoolToEventsDH) = (elit_X);
        b1 := b1 AND (NOT(ivar_s_xpos_at1));
        b1 := b1 AND ((state0.dvar_M_sup_S_xpos_at1) = (elit_On));
        IF b1 THEN
            progress := TRUE;
            state1 := state0;

            state1.dvar_M_sup_S_xpos_at1 := elit_Off;

            state0 := state1;
        END_IF;
    END_IF;

    // Event "S_xpos_at1_u_on".
    IF NOT progress THEN
        b1 := (state0.dvar_M_BoolToEventsDH) = (elit_X);
        b1 := b1 AND (ivar_s_xpos_at1);
        b1 := b1 AND ((state0.dvar_M_sup_HDynamics1) = (elit_X));
        b1 := b1 AND ((state0.dvar_M_sup_S_xpos_at2) = (elit_Off));
        b1 := b1 AND ((state0.dvar_M_sup_S_xpos_at3) = (elit_Off));
        b1 := b1 AND ((state0.dvar_M_sup_S_xpos_atdrop) = (elit_Off));
        b1 := b1 AND ((state0.dvar_M_sup_S_xpos_at1) = (elit_Off));
        IF b1 THEN
            progress := TRUE;
            state1 := state0;

            state1.dvar_M_sup_S_xpos_at1 := elit_On;

            state0 := state1;
        END_IF;
    END_IF;

    // Event "S_xpos_at2_u_off".
    IF NOT progress THEN
        b1 := (state0.dvar_M_BoolToEventsDH) = (elit_X);
        b1 := b1 AND (NOT(ivar_s_xpos_at2));
        b1 := b1 AND ((state0.dvar_M_sup_S_xpos_at2) = (elit_On));
        IF b1 THEN
            progress := TRUE;
            state1 := state0;

            state1.dvar_M_sup_S_xpos_at2 := elit_Off;

            state0 := state1;
        END_IF;
    END_IF;

    // Event "S_xpos_at2_u_on".
    IF NOT progress THEN
        b1 := (state0.dvar_M_BoolToEventsDH) = (elit_X);
        b1 := b1 AND (ivar_s_xpos_at2);
        b1 := b1 AND ((state0.dvar_M_sup_HDynamics1) = (elit_X));
        b1 := b1 AND ((state0.dvar_M_sup_S_xpos_at1) = (elit_Off));
        b1 := b1 AND ((state0.dvar_M_sup_S_xpos_at3) = (elit_Off));
        b1 := b1 AND ((state0.dvar_M_sup_S_xpos_atdrop) = (elit_Off));
        b1 := b1 AND ((state0.dvar_M_sup_S_xpos_at2) = (elit_Off));
        IF b1 THEN
            progress := TRUE;
            state1 := state0;

            state1.dvar_M_sup_S_xpos_at2 := elit_On;

            state0 := state1;
        END_IF;
    END_IF;

    // Event "S_xpos_at3_u_off".
    IF NOT progress THEN
        b1 := (state0.dvar_M_BoolToEventsDH) = (elit_X);
        b1 := b1 AND (NOT(ivar_s_xpos_at3));
        b1 := b1 AND ((state0.dvar_M_sup_S_xpos_at3) = (elit_On));
        IF b1 THEN
            progress := TRUE;
            state1 := state0;

            state1.dvar_M_sup_S_xpos_at3 := elit_Off;

            state0 := state1;
        END_IF;
    END_IF;

    // Event "S_xpos_at3_u_on".
    IF NOT progress THEN
        b1 := (state0.dvar_M_BoolToEventsDH) = (elit_X);
        b1 := b1 AND (ivar_s_xpos_at3);
        b1 := b1 AND ((state0.dvar_M_sup_HDynamics1) = (elit_X));
        b1 := b1 AND ((state0.dvar_M_sup_S_xpos_at1) = (elit_Off));
        b1 := b1 AND ((state0.dvar_M_sup_S_xpos_at2) = (elit_Off));
        b1 := b1 AND ((state0.dvar_M_sup_S_xpos_atdrop) = (elit_Off));
        b1 := b1 AND ((state0.dvar_M_sup_S_xpos_at3) = (elit_Off));
        IF b1 THEN
            progress := TRUE;
            state1 := state0;

            state1.dvar_M_sup_S_xpos_at3 := elit_On;

            state0 := state1;
        END_IF;
    END_IF;

    // Event "S_xpos_atdrop_u_off".
    IF NOT progress THEN
        b1 := (state0.dvar_M_BoolToEventsDH) = (elit_X);
        b1 := b1 AND (NOT(ivar_s_xpos_atdrop));
        b1 := b1 AND ((state0.dvar_M_sup_S_xpos_atdrop) = (elit_On));
        IF b1 THEN
            progress := TRUE;
            state1 := state0;

            state1.dvar_M_sup_S_xpos_atdrop := elit_Off;

            state0 := state1;
        END_IF;
    END_IF;

    // Event "S_xpos_atdrop_u_on".
    IF NOT progress THEN
        b1 := (state0.dvar_M_BoolToEventsDH) = (elit_X);
        b1 := b1 AND (ivar_s_xpos_atdrop);
        b1 := b1 AND ((state0.dvar_M_sup_HDynamics1) = (elit_X));
        b1 := b1 AND ((state0.dvar_M_sup_S_xpos_at1) = (elit_Off));
        b1 := b1 AND ((state0.dvar_M_sup_S_xpos_at2) = (elit_Off));
        b1 := b1 AND ((state0.dvar_M_sup_S_xpos_at3) = (elit_Off));
        b1 := b1 AND ((state0.dvar_M_sup_S_xpos_atdrop) = (elit_Off));
        IF b1 THEN
            progress := TRUE;
            state1 := state0;

            state1.dvar_M_sup_S_xpos_atdrop := elit_On;

            state0 := state1;
        END_IF;
    END_IF;

    // Event "S_zpos_atdown_u_off".
    IF NOT progress THEN
        b1 := (state0.dvar_M_BoolToEventsDH) = (elit_X);
        b1 := b1 AND (NOT(ivar_s_zpos_atdown));
        b1 := b1 AND ((state0.dvar_M_sup_S_zpos_atdown) = (elit_On));
        IF b1 THEN
            progress := TRUE;
            state1 := state0;

            state1.dvar_M_sup_S_zpos_atdown := elit_Off;

            state0 := state1;
        END_IF;
    END_IF;

    // Event "S_zpos_atdown_u_on".
    IF NOT progress THEN
        b1 := (state0.dvar_M_BoolToEventsDH) = (elit_X);
        b1 := b1 AND (ivar_s_zpos_atdown);
        b1 := b1 AND ((state0.dvar_M_sup_HDynamics3) = (elit_X));
        b1 := b1 AND ((state0.dvar_M_sup_S_zpos_atup) = (elit_Off));
        b1 := b1 AND ((state0.dvar_M_sup_S_zpos_atdown) = (elit_Off));
        IF b1 THEN
            progress := TRUE;
            state1 := state0;

            state1.dvar_M_sup_S_zpos_atdown := elit_On;

            state0 := state1;
        END_IF;
    END_IF;

    // Event "S_zpos_atup_u_off".
    IF NOT progress THEN
        b1 := (state0.dvar_M_BoolToEventsDH) = (elit_X);
        b1 := b1 AND (NOT(ivar_s_zpos_atup));
        b1 := b1 AND ((state0.dvar_M_sup_S_zpos_atup) = (elit_On));
        IF b1 THEN
            progress := TRUE;
            state1 := state0;

            state1.dvar_M_sup_S_zpos_atup := elit_Off;

            state0 := state1;
        END_IF;
    END_IF;

    // Event "S_zpos_atup_u_on".
    IF NOT progress THEN
        b1 := (state0.dvar_M_BoolToEventsDH) = (elit_X);
        b1 := b1 AND (ivar_s_zpos_atup);
        b1 := b1 AND ((state0.dvar_M_sup_HDynamics3) = (elit_X));
        b1 := b1 AND ((state0.dvar_M_sup_S_zpos_atdown) = (elit_Off));
        b1 := b1 AND ((state0.dvar_M_sup_S_zpos_atup) = (elit_Off));
        IF b1 THEN
            progress := TRUE;
            state1 := state0;

            state1.dvar_M_sup_S_zpos_atup := elit_On;

            state0 := state1;
        END_IF;
    END_IF;

    // Event "STimer_c_on".
    IF NOT progress THEN
        b1 := (state0.dvar_M_STimer1) = (elit_Off);
        b1 := b1 AND ((state0.dvar_M_sup_STimer) = (elit_Off));
        b1 := b1 AND ((state0.dvar_M_sup_sup) = (elit_X));
        b1 := b1 AND ((state0.dvar_M_sup_S_product) = (elit_On));
        IF b1 THEN
            progress := TRUE;
            state1 := state0;

            state1.dvar_M_STimer1 := elit_Running;
            state1.dvar_M_sup_STimer := elit_Running;

            state0 := state1;
        END_IF;
    END_IF;

    // Event "STimer_c_reset".
    IF NOT progress THEN
        b2 := (state0.dvar_M_STimer1) = (elit_Running);
        b2 := b2 OR ((state0.dvar_M_STimer1) = (elit_Timeout));
        b1 := b2;
        IF b1 THEN
            b2 := (state0.dvar_M_sup_STimer) = (elit_Running);
            b2 := b2 OR ((state0.dvar_M_sup_STimer) = (elit_Timeout));
            b1 := b1 AND (b2);
        END_IF;
        b1 := b1 AND ((state0.dvar_M_sup_sup) = (elit_X));
        b1 := b1 AND ((state0.dvar_M_sup_S_slidefull) = (elit_On));
        IF b1 THEN
            progress := TRUE;
            state1 := state0;

            IF ((state0.dvar_M_STimer1) = (elit_Running)) THEN
                state1.cvar_M_STimer1_t := 0.0;
                state1.dvar_M_STimer1 := elit_Off;
            ELSIF ((state0.dvar_M_STimer1) = (elit_Timeout)) THEN
                state1.cvar_M_STimer1_t := 0.0;
                state1.dvar_M_STimer1 := elit_Off;
            END_IF;
            IF ((state0.dvar_M_sup_STimer) = (elit_Running)) THEN
                state1.dvar_M_sup_STimer := elit_Off;
            ELSIF ((state0.dvar_M_sup_STimer) = (elit_Timeout)) THEN
                state1.dvar_M_sup_STimer := elit_Off;
            END_IF;

            state0 := state1;
        END_IF;
    END_IF;

    // Event "STimer_u_timeout".
    IF NOT progress THEN
        b1 := (state0.dvar_M_STimer1) = (elit_Running);
        b1 := b1 AND ((state0.cvar_M_STimer1_t) > (0.5));
        b1 := b1 AND ((state0.dvar_M_sup_STimer) = (elit_Running));
        IF b1 THEN
            progress := TRUE;
            state1 := state0;

            state1.dvar_M_STimer1 := elit_Timeout;
            state1.dvar_M_sup_STimer := elit_Timeout;

            state0 := state1;
        END_IF;
    END_IF;

    // Event "Timer_c_on".
    IF NOT progress THEN
        b1 := (state0.dvar_M_sup_sup) = (elit_X);
        b1 := b1 AND ((state0.dvar_M_sup_S_turntable) = (elit_On));
        b1 := b1 AND ((state0.dvar_M_sup_Timer) = (elit_Off));
        b1 := b1 AND ((state0.dvar_M_Timer1) = (elit_Off));
        IF b1 THEN
            progress := TRUE;
            state1 := state0;

            state1.dvar_M_sup_Timer := elit_Running;
            state1.dvar_M_Timer1 := elit_Running;

            state0 := state1;
        END_IF;
    END_IF;

    // Event "Timer_c_reset".
    IF NOT progress THEN
        b1 := (state0.dvar_M_sup_sup) = (elit_X);
        b1 := b1 AND ((state0.dvar_M_sup_S_turntable) = (elit_Off));
        IF b1 THEN
            b2 := (state0.dvar_M_sup_Timer) = (elit_Running);
            b2 := b2 OR ((state0.dvar_M_sup_Timer) = (elit_Timeout));
            b1 := b1 AND (b2);
        END_IF;
        IF b1 THEN
            b2 := (state0.dvar_M_Timer1) = (elit_Running);
            b2 := b2 OR ((state0.dvar_M_Timer1) = (elit_Timeout));
            b1 := b1 AND (b2);
        END_IF;
        IF b1 THEN
            progress := TRUE;
            state1 := state0;

            IF ((state0.dvar_M_sup_Timer) = (elit_Running)) THEN
                state1.dvar_M_sup_Timer := elit_Off;
            ELSIF ((state0.dvar_M_sup_Timer) = (elit_Timeout)) THEN
                state1.dvar_M_sup_Timer := elit_Off;
            END_IF;
            IF ((state0.dvar_M_Timer1) = (elit_Running)) THEN
                state1.cvar_M_Timer1_t := 0.0;
                state1.dvar_M_Timer1 := elit_Off;
            ELSIF ((state0.dvar_M_Timer1) = (elit_Timeout)) THEN
                state1.cvar_M_Timer1_t := 0.0;
                state1.dvar_M_Timer1 := elit_Off;
            END_IF;

            state0 := state1;
        END_IF;
    END_IF;

    // Event "Timer_u_timeout".
    IF NOT progress THEN
        b1 := (state0.dvar_M_sup_Timer) = (elit_Running);
        b1 := b1 AND ((state0.dvar_M_Timer1) = (elit_Running));
        b1 := b1 AND ((state0.cvar_M_Timer1_t) > (0.5));
        IF b1 THEN
            progress := TRUE;
            state1 := state0;

            state1.dvar_M_sup_Timer := elit_Timeout;
            state1.dvar_M_Timer1 := elit_Timeout;

            state0 := state1;
        END_IF;
    END_IF;

    // Event "TTimer_c_on".
    IF NOT progress THEN
        b1 := (state0.dvar_M_sup_sup) = (elit_X);
        IF b1 THEN
            b3 := (state0.dvar_M_sup_A_elevator_down) = (elit_On);
            b3 := b3 AND ((state0.dvar_M_sup_S_Tinitialized) = (elit_On));
            b2 := b3;
            IF NOT(b2) THEN
                b3 := (state0.dvar_M_sup_A_elevator_down) = (elit_Off);
                IF b3 THEN
                    b4 := (state0.dvar_M_sup_PusherLift) = (elit_Two);
                    b4 := b4 OR ((state0.dvar_M_sup_PusherLift) = (elit_Four));
                    b3 := b3 AND (b4);
                END_IF;
                b3 := b3 AND ((state0.dvar_M_sup_S_Tinitialized) = (elit_On));
                b2 := b2 OR (b3);
            END_IF;
            b1 := b1 AND (b2);
        END_IF;
        b1 := b1 AND ((state0.dvar_M_sup_TTimer) = (elit_Off));
        b1 := b1 AND ((state0.dvar_M_TTimer1) = (elit_Off));
        IF b1 THEN
            progress := TRUE;
            state1 := state0;

            state1.dvar_M_sup_TTimer := elit_Running;
            state1.dvar_M_TTimer1 := elit_Running;

            state0 := state1;
        END_IF;
    END_IF;

    // Event "TTimer_c_reset".
    IF NOT progress THEN
        b1 := (state0.dvar_M_sup_sup) = (elit_X);
        b1 := b1 AND ((state0.dvar_M_sup_A_elevator_down) = (elit_Off));
        IF b1 THEN
            b2 := (state0.dvar_M_sup_PusherLift) = (elit_One);
            b2 := b2 OR ((state0.dvar_M_sup_PusherLift) = (elit_Three));
            b1 := b1 AND (b2);
        END_IF;
        b1 := b1 AND ((state0.dvar_M_sup_S_Tinitialized) = (elit_On));
        IF b1 THEN
            b2 := (state0.dvar_M_sup_TTimer) = (elit_Running);
            b2 := b2 OR ((state0.dvar_M_sup_TTimer) = (elit_Timeout));
            b1 := b1 AND (b2);
        END_IF;
        IF b1 THEN
            b2 := (state0.dvar_M_TTimer1) = (elit_Running);
            b2 := b2 OR ((state0.dvar_M_TTimer1) = (elit_Timeout));
            b1 := b1 AND (b2);
        END_IF;
        IF b1 THEN
            progress := TRUE;
            state1 := state0;

            IF ((state0.dvar_M_sup_TTimer) = (elit_Running)) THEN
                state1.dvar_M_sup_TTimer := elit_Off;
            ELSIF ((state0.dvar_M_sup_TTimer) = (elit_Timeout)) THEN
                state1.dvar_M_sup_TTimer := elit_Off;
            END_IF;
            IF ((state0.dvar_M_TTimer1) = (elit_Running)) THEN
                state1.cvar_M_TTimer1_t := 0.0;
                state1.dvar_M_TTimer1 := elit_Off;
            ELSIF ((state0.dvar_M_TTimer1) = (elit_Timeout)) THEN
                state1.cvar_M_TTimer1_t := 0.0;
                state1.dvar_M_TTimer1 := elit_Off;
            END_IF;

            state0 := state1;
        END_IF;
    END_IF;

    // Event "TTimer_u_timeout".
    IF NOT progress THEN
        b1 := (state0.dvar_M_sup_TTimer) = (elit_Running);
        b1 := b1 AND ((state0.dvar_M_TTimer1) = (elit_Running));
        b1 := b1 AND ((state0.cvar_M_TTimer1_t) > (0.5));
        IF b1 THEN
            progress := TRUE;
            state1 := state0;

            state1.dvar_M_sup_TTimer := elit_Timeout;
            state1.dvar_M_TTimer1 := elit_Timeout;

            state0 := state1;
        END_IF;
    END_IF;

    // Event "tau".
    IF NOT progress THEN
        b1 := (state0.dvar_M_HardwareMapDH) = (elit_init0);
        b1 := b1 AND ((state0.cvar_M_HardwareMapDH_t) >= (2.0));
        IF b1 THEN
            progress := TRUE;
            state1 := state0;

            state1.dvar_M_HardwareMapDH := elit_init1;

            state0 := state1;
        END_IF;
    END_IF;

    // Event "tau".
    IF NOT progress THEN
        IF (state0.dvar_M_HardwareMapDH) = (elit_init1) THEN
            progress := TRUE;
            state1 := state0;

            state1.dvar_M_HardwareMapDH_out_a_x2testing := FALSE;
            state1.dvar_M_HardwareMapDH := elit_init2;

            state0 := state1;
        END_IF;
    END_IF;

    // Event "tau".
    IF NOT progress THEN
        b1 := (state0.dvar_M_HardwareMapDH) = (elit_init2);
        IF b1 THEN
            b2 := ivar_s_xpos_at1;
            b2 := b2 OR (ivar_s_xpos_at2);
            b1 := b1 AND (b2);
        END_IF;
        IF b1 THEN
            progress := TRUE;
            state1 := state0;

